# B&R Automation Studio project IecStringPrj
Automation Studio 4.11.5.46 SP; Sample project and development for IecString library

## Configuration ARM

CPU X20CP0484, AutomationRuntime 6.3.4, Build 11.3.0

### Task classes (Cpu.sw)
```
Libraries: IecString, AsBrStr, astime, runtime
```

### Hardware
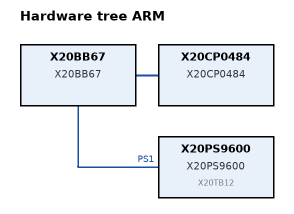
```
X20BB67 : X20BB67 v1.3.1.0
X20CP0484 : X20CP0484 v1.8.1.0  [SL -> X20BB67.SL1]
  Connector IF2:
    ActivateDevice = 1
    InaPort = 11160
  ConfigurationID = IecStringProject_ARM
  UserPartitionSize = 0
  TimerDeviceType = SWIOTIMER
  Cyclic1Duration = 10000
  Cyclic1Tolerance = 10000
  Cyclic2Duration = 20000
  Cyclic2Tolerance = 20000
  Cyclic3Duration = 50000
  Cyclic3Tolerance = 50000
  Cyclic4Duration = 100000
  Cyclic4Tolerance = 100000
  Cyclic5Duration = 200000
  Cyclic5Tolerance = 200000
  Cyclic6Duration = 500000
  Cyclic6Tolerance = 500000
  Cyclic7Duration = 1000000
  Cyclic7Tolerance = 1000000
  Cyclic8Duration = 10000
  Cyclic8Tolerance = 30000000
  FileDevice1
  FileDeviceName1 = USER
  FileDevicePath1 = USER_PATH
  ActivateFtpServer = 1
  ActivateWebServer = 1
  ActivateSdm = 1
X20PS9600 : X20PS9600 v1.6.2.0  [PS -> X20BB67.PS1; SS1 -> X20TB12.SS]
X20TB12 : X20TB12 v1.0.0.0
```

## Configuration ARsim

CPU PC_any, AutomationRuntime B4.73, Build 4.1.2, Vc V4.72.2

### Task classes (Cpu.sw)
```
Cyclic#1:
  Sample <- Sample.prg
Binaries: FWRules, TCData, udbdef, asfw, User, iomap, sysconf, arconfig, ashwd, Role, ashwac
Libraries: BRSE_ARL, AsBrStr, ArEventLog, sys_lib, runtime, asieccon, astime, IecFrmtStr
```

## Configuration Hardware

CPU X20CP1585, AutomationRuntime E4.92, Build 6.3.0

### Task classes (Cpu.sw)
```
Cyclic#1:
  ACopy1C <- Source.Performance.ACopy1C.prg
  ACopy2Iec <- Source.Performance.ACopy2Iec.prg
  ACopy3Brs <- Source.Performance.ACopy3Brs.prg
  ACopy4Lib <- Source.Performance.ACopy4Lib.prg
  PerfCCopy <- (binary)
  PerfBrCopy <- (binary)
  PerfISDec <- (binary)
  PerfBrDec <- (binary)
  PerfISCopy <- (binary)
Libraries: IecString, AsBrStr, astime, runtime
```

### Hardware
```
X20CP1585 : X20CP1585 v1.10.0.0
  Connector IF1:
    ActivateIna = 0
  Connector IF2:
    ActivateDevice = 1
    HostName = chicago-x20cp1585
  Connector IF3:
    EplHostName = chicago-x20cp1585
    HostName = chicago-x20cp1585
  ConfigurationID = IecStringProject_Hardware
  FileDevice1
  FileDeviceName1 = USER
  FileDevicePath1 = USER_PATH
  EthernetHostName = chicago-x20cp1585
```

## Configuration IA32

CPU X20CP1685, AutomationRuntime 6.3.4, Build 11.3.0, Vc 

### Task classes (Cpu.sw)
```
Libraries: IecString
```

### Hardware
```
X20CP1685 : X20CP1685 v1.8.1.0
  FileDevice1
  FileDeviceName1 = USER
  FileDevicePath1 = USER_PATH
```

## Configuration Intel

CPU X20CP1586, AutomationRuntime E4.92, Build 6.3.0

### Task classes (Cpu.sw)
```
Cyclic#1:
  PerfCCopy <- (binary)
  PerfBrCopy <- (binary)
  PerfISDec <- (binary)
  PerfBrDec <- (binary)
  PerfISCopy <- (binary)
Binaries: TCData, udbdef, asfw, sysconf, arconfig, ashwd, ashwac
Libraries: IecString, astime, standard, asieccon
```

### Hardware
```
X20CP1586 : X20CP1586 v1.10.0.0
  Connector IF1:
    ActivateIna = 0
  Connector IF2:
    ActivateDevice = 1
  ConfigurationID = IecStringProject_Intel
  FileDevice1
  FileDeviceName1 = USER
  FileDevicePath1 = USER_PATH
```

## Configuration Simulation

CPU PC_any, AutomationRuntime C4.90, Build 4.1.2, Vc 

### Task classes (Cpu.sw)
```
Cyclic#1:
  Sample <- Sample.prg
  CUsage <- CUsage.prg
Binaries: FWRules, TCData, udbdef, asfw, User, iomap, sysconf, arconfig, ashwd, Role, ashwac
Libraries: AsBrStr, runtime, IecString, asieccon, astime
```

### Hardware
```
X20CP1586 : X20CP1586 v1.10.0.0
  Connector IF1:
    ActivateIna = 0
  Connector IF2:
    ActivateDevice = 1
    InaPort = 11160
  ConfigurationID = IecStringPrj_Simulation
```

## Configuration UnitTest

CPU PC_any, AutomationRuntime 6.3.4, Build 11.3.0

### Task classes (Cpu.sw)
```
Cyclic#1 (cycle 1000 us):
  TestSuite <- Source.UnitTest.TestSuite.prg
  ExSplit <- Source.Example.ExSplit.prg
Binaries: udbdef, TCData, sysconf, ashwd, asfw, arconfig, ashwac
Libraries: IecString, runtime, astime, UnitTest, UtMgr, sys_lib, UtWs, AsIecCon, AsBrStr
```

### Hardware
```
PC : PC_any v1.1.2.0 (OrderNumber=PC)
  ConfigurationID = IecStringProject_UnitTest
  SystemTick = 1000
  Cyclic1Duration = 1000
  FileDevice1
  FileDeviceName1 = USER
  FileDevicePath1 = USER_PATH
  ActivateFtpServer = 1
  ActivateWebServer = 1
  WebServerProtocol = 1
  ActivateSdm = 1
```

## Configuration X20CPU

CPU X20CP1585, AutomationRuntime E4.92, Build 6.3.0

CPU X20CP1586, AutomationRuntime E4.92, Build 4.1.2, Vc 

### Task classes (Cpu.sw)
```
Cyclic#1:
  CPUCopy <- Source.Performance.CPUCopy.prg
Cyclic#4:
  TestSuite <- Source.UnitTest.TestSuite.prg
  IECST <- Source.Sample.IECST.prg
  TestCStr <- Source.Compare.TestCStr.prg
Libraries: AsBrStr, IecString, UnitTest, UtMgr, UtWs, AsARCfg, runtime, AsIecCon, astime, sys_lib
```

### Task classes (Cpu.sw)
```
Cyclic#4:
  TestSuite <- TestSuite.prg
  IECST <- IECST.prg
Libraries: AsBrStr, IecString, UnitTest, UtMgr, UtWs, AsARCfg, runtime, AsIecCon, astime, sys_lib
```

### Hardware
```
X20CP1585 : X20CP1585 v1.10.0.0
  Connector IF1:
    ActivateIna = 0
  Connector IF2:
    ActivateDevice = 1
    HostName = chicago-x20cp1585
    InaPort = 11160
  Connector IF3:
    EplHostName = chicago-x20cp1585
    HostName = chicago-x20cp1585
  ConfigurationID = IecStringProject_X20CPU
  FileDevice1
  FileDeviceName1 = USER
  FileDevicePath1 = USER_PATH
  EthernetHostName = chicago-x20cp1585
```

## Logical view

Binary libraries used (declarations not repeated): IecString, UnitTest, UtMgr, UtWs, runtime, sys_lib, astime, AsBrStr, standard, AsIecCon

### Package Logical/Libraries - Global libraries

### Library Logical/Libraries/BRSE_ARL (ANSIC, version 2.00.0)
Depends on: AsBrStr, SYS_Lib, ArEventLog

#### BRSE_ARL.fun
```iecst
FUNCTION BRSE_ARL_Alloc : UINT (*Allocates the FIFO buffer for the logger*)
	VAR_INPUT
		ID : UINT; (*Logger ID of the logbook to be written to*)
		Name : STRING[25]; (*Name of the logbook to which to write to.*)
		LogbookSize : UDINT; (*Size of the logbook in bytes (if a new one has to be created).*)
		MessageSize : UDINT; (*Maximum length of a single message string for the logbook*)
		BufferedEntries : UDINT; (*Maximum number of messages that can be stored in the FIFO buffer*)
	END_VAR
END_FUNCTION
(*	VAR_INPUT
		ID : UINT; (*Logger ID of the logbook to be written to*)
(*		ErrorNumber : UDINT; (*Error number to show up in the logbook*)
(*FUNCTION BRSE_ARL_Info : UINT (*Writes an info message to the logbook*)
(*		ErrorMessage : STRING[32767]; (*Error message in the logbook*)
(*		pMsgData : UDINT; (*Address of a BRSE_ARL_Arguments_typ structure that contains data values*)
(*	END_VAR
END_FUNCTION--*/ *)

FUNCTION BRSE_ARL_Cyclic : DINT (*Cyclic call to flush pending entries to the logbook*)
	VAR_INPUT
		ID : UINT; (*Logger ID of the logbook to be written to*)
	END_VAR
END_FUNCTION

FUNCTION_BLOCK BRSE_ARL_DebugInfo
	VAR_INPUT
		ID : UINT;
	END_VAR
	VAR_OUTPUT
		Info : BRSE_ARL_Logger_typ;
		Status : UINT;
	END_VAR
END_FUNCTION_BLOCK
(*FUNCTION BRSE_ARL_Fatal : UINT (*Writes a fatal message to the logbook*)
(*	VAR_INPUT
				ID : UINT; (*Logger ID of the logbook to be written to*)
(*		ErrorNumber : UDINT; (*Error number to show up in the logbook*)
(*		ErrorMessage : STRING[32767]; (*Error message in the logbook*)
(*		pMsgData : UDINT; (*Address of a BRSE_ARL_Arguments_typ structure that contains data values*)
(*	END_VAR
(*END_FUNCTION *)

FUNCTION BRSE_ARL_Free : UINT (*Deallocates the FIFO buffer *)
	VAR_INPUT
		ID : UINT; (*Logger ID of the logbook to be written to*)
	END_VAR
END_FUNCTION
(*FUNCTION BRSE_ARL_Warning : UINT (*Writes a warning message to the logbook*)
(*	VAR_INPUT
		ID : UINT; (*Logger ID of the logbook to be written to*)
(*		ErrorNumber : UDINT; (*Error number to show up in the logbook*)
(*		ErrorMessage : STRING[32767]; (*Error message in the logbook*)
(*		pMsgData : UDINT; (*Address of a BRSE_ARL_Arguments_typ structure that contains data values*)
(*	END_VAR
(*END_FUNCTION*)

FUNCTION BRSE_ARL_Log : UINT
	VAR_INPUT
		ID : UINT;
		ErrorNumber : UDINT;
		User : STRING[32];
		ErrorMessage : STRING[32767];
	END_VAR
END_FUNCTION
```

#### BRSE_ARL.typ
```iecst
TYPE
	BRSE_ARL_Arguments_typ : 	STRUCT
		r : ARRAY[0..4]OF REAL;
		s : ARRAY[0..4]OF UDINT;
		b : ARRAY[0..4]OF BOOL;
		i : ARRAY[0..4]OF DINT;
	END_STRUCT;
	BRSE_ARL_Logger_typ : 	STRUCT  (* ID CHECK *)
		ID : UDINT; (*unsigned long ID;*) (*Size of the structure*)
		LoggerTypSize : DINT; (*long LoggerTypSize;*) (*VARIABLES*)
		LogbookIdent : UDINT; (*UDINT LogbookIdent;*)
		LogbookSize : UDINT; (*UDINT LogbookSize;*) (*Size of the logbook*)
		LogbookName : STRING[26]; (*char LogbookName[26];*) (*Name of the logbook (max. 25 chars)*)
		MaxMessageSize : UDINT; (*unsigned int MaxMessageSize;*) (*Max. size of a text message*)
		Cyclic_Step : UDINT; (*unsigned int Cyclic_Step;*) (* FUNCTION BLOCKS *)
		FB_ArEventLogGetIdent : ArEventLogGetIdent; (*AsArLogGetInfo_typ FB_AsArLogGetInfo;*)
		FB_ArEventLogCreate : ArEventLogCreate; (*AsArLogCreate_typ  FB_AsArLogCreate;*)
		FB_ArEventLogWrite : ArEventLogWrite; (*AsArLogWrite_typ   FB_AsArLogWrite;*) (*FIFO BUFFER*)
		fifo_write_lock : BOOL; (*Locks critical sections in the FIFO write processing*)
		fifo_reset : BOOL; (*Clearing FIFO memory, used if FIFO full when trying to read.*)
		tempString : STRING[50];
		EntrySize : UDINT; (* Size of a single logbook entry *)
		MaxBufEntries : UDINT; (*Max. number of buffered entries*)
		CurBufEntries : UDINT; (*Number of entries in the buffer*)
		ReadIndex : UDINT; (*Current index from which to read*)
		WriteIndex : UDINT; (* Current index at which to write *)
		Buffer : ARRAY[0..0]OF BRSE_ARL_LogbookEntry_typ; (*Buffer start position (must be last in the struct)*)
	END_STRUCT;
	BRSE_ARL_LogbookEntry_typ : 	STRUCT
		User : STRING[36];
		ErrorNo : UDINT;
		ErrorMsg : STRING[0]; (* Only buffer start position, size depends on the requested size in Alloc *)
	END_STRUCT;
END_TYPE
```

#### brse_arl_alloc.c
```c
/*! \file brse_arl_alloc.c */

#include "brse_arl_main.h"

/* List of all available loggers */
BRSE_ARL_Logger_typ* BRSE_ARL_LoggerList[BRSE_ARL_MAX_LOGGERS];

/*! \interface BRSE_ARL_Alloc
	\brief Allocates the FIFO buffer for the logger

	This function allocates a FIFO buffer of the given size to be used for further
	buffered logbook writing functions. It also takes parameters that will be used in \ref BRSE_ARL_Cyclic().
	NOTE: Should be called in the _INIT part of a task!

	The following is done in \ref BRSE_ARL_Cyclic(): If logbook does not exist a new one will be created with the supplied name.
	If no name has been supplied, the default user logbook will be used.

	\param ID Logger ID of the logbook to be written to
    \param Name Name of the logbook to which to write to.
    \param LogbookSize Size of the logbook in bytes (if a new one has to be created). Note: at least 4096
    \param MessageSize Maximum length of a single message string for the logbook
    \param BufferedEntries Maximum number of messages that can be stored in the FIFO buffer
    \retval \c 0 Function call successful
*/
unsigned short BRSE_ARL_Alloc(unsigned short ID, plcstring* Name, unsigned long LogbookSize, unsigned long MessageSize, unsigned long BufferedEntries)
{
	BRSE_ARL_Logger_typ* pLogger;
	unsigned long EntrySize;
	unsigned long LoggerTypSize;

	/* Check if ID is in range */
	if (ID >= BRSE_ARL_MAX_LOGGERS)
	{
		return BRSE_ARL_ID_NOT_VALID;
	}

	/* Access the chosen logger */
	pLogger = BRSE_ARL_LoggerList[ID];

	/* Check, if ID is valid */
	if ((pLogger != NULL) && (pLogger->ID == (BRSE_ARL_ID_BASE | (unsigned long)ID)))
	{
		return BRSE_ARL_ID_ALREADY_INITIALIZED;
	}

	/* ID is not used yet, so allocate memory for it */

	/* Calculate the entry size and the logger size */
	EntrySize = (unsigned long)sizeof(BRSE_ARL_LogbookEntry_typ) + MessageSize + 1;
	LoggerTypSize = (unsigned long)sizeof(BRSE_ARL_Logger_typ) + BufferedEntries * EntrySize;

	/* Allocate memory for the logger */
	if (TMP_alloc(LoggerTypSize, (void**)&pLogger) != 0)
	{
		/* Memory allocation failed */
		return BRSE_ARL_OUT_OF_MEMORY;
	}
	/* Put valid information into the logger structure */
	memset((void*)pLogger, 0, LoggerTypSize);

	/* Store some information */
	pLogger->ID = BRSE_ARL_ID_BASE | (unsigned long)ID;
	pLogger->LoggerTypSize = LoggerTypSize;

	strncpy(pLogger->LogbookName, Name, sizeof(pLogger->LogbookName));
	pLogger->LogbookSize = LogbookSize;
	pLogger->MaxMessageSize = MessageSize;
	pLogger->EntrySize = EntrySize;
	pLogger->MaxBufEntries = BufferedEntries;

	/* Save the new logger */
	BRSE_ARL_LoggerList[ID] = pLogger;

	return ERR_OK;
}

/*! \interface BRSE_ARL_Free
	\brief Deallocates the FIFO buffer

	This function writes all pending entries to the logbook and closes down the buffer.
	NOTE: Not to be called in the cyclic part of a task!

	\param ID Logger ID of the logbook to be written to
    \return \c 0 Function call successful
*/
unsigned short BRSE_ARL_Free(unsigned short ID)
{
	/* Check if ID is valid */
	if ((ID >= BRSE_ARL_MAX_LOGGERS)
		|| (BRSE_ARL_LoggerList[ID] == NULL)
		|| (BRSE_ARL_LoggerList[ID]->ID != (BRSE_ARL_ID_BASE | (unsigned long)ID)))
	{
		return BRSE_ARL_ID_NOT_VALID;
	}

	/* Flush pending writes */
	while (BRSE_ARL_Cyclic(ID) == 65535);

	/* Release allocated memory */
	TMP_free(BRSE_ARL_LoggerList[ID]->LoggerTypSize, (void*)BRSE_ARL_LoggerList[ID]);
	BRSE_ARL_LoggerList[ID] = NULL;

	return ERR_OK;
}
```

#### brse_arl_cyclic.c
```c
/*! \file brse_arl_cyclic.c */

#include "brse_arl_main.h"

/*! \interface BRSE_ARL_Cyclic
	\brief Cyclic call to flush pending entries to the logbook

	This function writes pending entries to the logbook and has to be called cyclically.

	\param ID Logger ID of the logbook to be written to
    \retval 0 all messages written to logger
	\retval 65535 pending entries to be written
	\retval Error Error code from the ArEventLog library
*/

long BRSE_ARL_Cyclic(unsigned short ID)
{
	BRSE_ARL_Logger_typ* pLogger = NULL;
	BRSE_ARL_LogbookEntry_typ* pCurEntry = NULL;
	DINT status = ERR_FUB_BUSY;

	/* Check if ID is valid */
	if ((ID >= BRSE_ARL_MAX_LOGGERS)
		|| (BRSE_ARL_LoggerList[ID] == NULL)
		|| (BRSE_ARL_LoggerList[ID]->ID != (BRSE_ARL_ID_BASE | (unsigned long)ID)))
	{
		return BRSE_ARL_ID_NOT_VALID;
	}

	/* Access the chosen logger */
	pLogger = BRSE_ARL_LoggerList[ID];

	switch (pLogger->Cyclic_Step)
	{
		/* Initialize */
		case 0:

			pLogger->Cyclic_Step = 1;

		/* GET LOGBOOK */
		case 1:
			/* Check if a logbook with the given name is existing */
			pLogger->FB_ArEventLogGetIdent.Execute = TRUE;
			strcpy(pLogger->FB_ArEventLogGetIdent.Name, pLogger->LogbookName);

			ArEventLogGetIdent(&pLogger->FB_ArEventLogGetIdent);

			if(pLogger->FB_ArEventLogGetIdent.Done)
			{
				/* Save the ident of the exisiting logbook */
				pLogger->LogbookIdent = pLogger->FB_ArEventLogGetIdent.Ident;

				/* Go to operating state */
				pLogger->Cyclic_Step = 10;
				status = ERR_FUB_BUSY;
			}
			else if(pLogger->FB_ArEventLogGetIdent.Error)
			{
				if(pLogger->FB_ArEventLogGetIdent.StatusID == arEVENTLOG_ERR_LOGBOOK_NOT_FOUND)
				{
					pLogger->Cyclic_Step = 2;
					status = ERR_FUB_BUSY;
				}
				else
				{
					status = pLogger->FB_ArEventLogGetIdent.StatusID;
				}
			}
			else
			{
				status = ERR_FUB_BUSY;
			}

			break;

		/* CREATE LOGBOOK */
		case 2:
			/* Create a new logbook in USRROM */
			pLogger->FB_ArEventLogCreate.Execute = TRUE;
			strcpy(pLogger->FB_ArEventLogCreate.Name, pLogger->LogbookName);
			pLogger->FB_ArEventLogCreate.Size = pLogger->LogbookSize;
			pLogger->FB_ArEventLogCreate.Persistence = arEVENTLOG_PERSISTENCE_PERSIST;

			ArEventLogCreate(&pLogger->FB_ArEventLogCreate);

			if(pLogger->FB_ArEventLogCreate.Done)
			{
				pLogger->LogbookIdent = pLogger->FB_ArEventLogCreate.Ident;

				/* Go to operating state */
				pLogger->Cyclic_Step = 10;
				status = ERR_FUB_BUSY;
			}
			else if(pLogger->FB_ArEventLogCreate.Busy)
			{
				status = ERR_FUB_BUSY;
			}
			else if(pLogger->FB_ArEventLogCreate.Error)
			{
				status = pLogger->FB_ArEventLogCreate.StatusID;
			}

			break;

		/* POP ENTRY FROM THE FIFO AND WRITE IT TO THE LOGBOOK */
		case 10:
			status = ERR_FUB_BUSY;
			if ( (pLogger->CurBufEntries == 0) )
			{
				/* No entry in the fifo */
				/* Answer with OK then... */
				status = ERR_OK;
			}
			else if (!pLogger->fifo_write_lock)
			{
				if ( (pLogger->CurBufEntries >= pLogger->MaxBufEntries) )
				{
					/*Lock the buffer directly to avoid loosing data*/
					pLogger->fifo_reset = 1;

					/*State change, prepare to reset buffer*/
					pLogger->Cyclic_Step = 14;

					status = ERR_FUB_BUSY;

				}
				else
				{
					/* Got an entry in the fifo */
					pCurEntry = (BRSE_ARL_LogbookEntry_typ*)((void*)pLogger->Buffer + pLogger->EntrySize * pLogger->ReadIndex);

					pLogger->FB_ArEventLogWrite.Execute = TRUE;
					pLogger->FB_ArEventLogWrite.Ident = pLogger->LogbookIdent;
					pLogger->FB_ArEventLogWrite.EventID = pCurEntry->ErrorNo;
					pLogger->FB_ArEventLogWrite.AddDataSize = strlen(pCurEntry->ErrorMsg) + 1;
					pLogger->FB_ArEventLogWrite.AddDataFormat = arEVENTLOG_ADDFORMAT_TEXT;
					pLogger->FB_ArEventLogWrite.AddData = (UDINT)pCurEntry->ErrorMsg;
					strcpy(pLogger->FB_ArEventLogWrite.ObjectID, pCurEntry->User);

					if(pLogger->FB_ArEventLogWrite.Done)
					{
						pLogger->FB_ArEventLogWrite.Execute = FALSE;
					}

					ArEventLogWrite(&pLogger->FB_ArEventLogWrite);

					if(pLogger->FB_ArEventLogWrite.Done)
					{
						pLogger->ReadIndex++;
						if (pLogger->ReadIndex >= pLogger->MaxBufEntries)
						{
							pLogger->ReadIndex = 0;
						}

						pLogger->CurBufEntries--;

						/* Return OK if no more entries shall be written */
						status = (pLogger->CurBufEntries == 0) ? ERR_OK : ERR_FUB_BUSY;
					}
					else if(pLogger->FB_ArEventLogWrite.Error)
					{
						status = pLogger->FB_ArEventLogWrite.StatusID;
					}
					else
					{
						status = ERR_FUB_BUSY;
					}
				}
			}
			else
			{
				/* Write is active */
				status = ERR_FUB_BUSY;
			}
			break;
		case 14:
			status = ERR_FUB_BUSY;

			if (pLogger->FB_ArEventLogWrite.StatusID == ERR_FUB_BUSY )
			{
				/*Wait if a line is being written to the logg book.*/
				ArEventLogWrite(&pLogger->FB_ArEventLogWrite);

			}
			else
			{

				/*Switch state, empty buffer.*/
				pLogger->Cyclic_Step = 15;
			}

			break;

		case 15: /*Output reset start message*/
				status = ERR_FUB_BUSY;

				pLogger->FB_ArEventLogWrite.Execute 		= TRUE;
				pLogger->FB_ArEventLogWrite.Ident 			= pLogger->LogbookIdent;
				pLogger->FB_ArEventLogWrite.EventID 		= -536820909; /* Severity = Error, Code = 50003 */
				strcpy(pLogger->tempString, "BUFFER RESET STARTED");
				pLogger->FB_ArEventLogWrite.AddData			= (UDINT)(pLogger->tempString);
				pLogger->FB_ArEventLogWrite.AddDataSize 	= strlen(pLogger->tempString) + 1;
				pLogger->FB_ArEventLogWrite.AddDataFormat 	= arEVENTLOG_ADDFORMAT_TEXT;

				ArEventLogWrite(&pLogger->FB_ArEventLogWrite);

				if (pLogger->FB_ArEventLogWrite.StatusID == ERR_OK )
				{
					/*Switch state, empty buffer.*/
					pLogger->Cyclic_Step = 20;

				}
			break;

		case 20: /*Empty the buffer, reset.*/
			status = ERR_FUB_BUSY;
			if ( (pLogger->CurBufEntries == 0) )
			{
				/*Buffer reset completed, switcht to state where message is output.*/
				pLogger->Cyclic_Step = 21;

			}
			else
			{
				/*Empty buffer*/
				/* Got an entry in the fifo */
				pCurEntry = (BRSE_ARL_LogbookEntry_typ*)((UDINT)pLogger->Buffer + pLogger->EntrySize * pLogger->ReadIndex);

				pLogger->FB_ArEventLogWrite.Execute 		= TRUE;
				pLogger->FB_ArEventLogWrite.Ident 			= pLogger->LogbookIdent;
				pLogger->FB_ArEventLogWrite.EventID 		= pCurEntry->ErrorNo;
				//TODO: Event ID log level
				pLogger->FB_ArEventLogWrite.AddDataFormat 	= arEVENTLOG_ADDFORMAT_TEXT;
				pLogger->FB_ArEventLogWrite.AddData 		= (UDINT)pCurEntry->ErrorMsg;
				strcpy(pLogger->FB_ArEventLogWrite.ObjectID, pCurEntry->User);
				//					pLogger->FB_AsArLogWrite.mem = (UDINT)NULL;
				//					pLogger->FB_AsArLogWrite.len = 0;

				ArEventLogWrite(&pLogger->FB_ArEventLogWrite);

				if(pLogger->FB_ArEventLogWrite.Done)
				{
					pLogger->ReadIndex++;
					if (pLogger->ReadIndex >= pLogger->MaxBufEntries)
					{
						pLogger->ReadIndex = 0;
					}

					pLogger->CurBufEntries--;

					/* Return OK if no more entries shall be written */
					status = (pLogger->CurBufEntries == 0) ? ERR_OK : ERR_FUB_BUSY;
				}
				else if(pLogger->FB_ArEventLogWrite.Error)
				{
					status = pLogger->FB_ArEventLogWrite.StatusID;
				}
				else
				{
					status = ERR_FUB_BUSY;
				}
			}
			break;

		case 21: /*Output message the reset is completed*/
				status = ERR_FUB_BUSY;

				pLogger->FB_ArEventLogWrite.Execute 		= TRUE;
				pLogger->FB_ArEventLogWrite.Ident 			= pLogger->LogbookIdent;
				pLogger->FB_ArEventLogWrite.EventID			= -536820908;
				pLogger->FB_ArEventLogWrite.AddDataFormat 	= arEVENTLOG_ADDFORMAT_TEXT;
				strcpy(pLogger->tempString, "BUFER RESET COMPLETED");
				pLogger->FB_ArEventLogWrite.AddData 		= (UDINT)pLogger->tempString;
				pLogger->FB_ArEventLogWrite.AddDataSize 	= strlen(pLogger->tempString) + 1;

				ArEventLogWrite(&pLogger->FB_ArEventLogWrite);

				status = ERR_FUB_BUSY;
				if (pLogger->FB_ArEventLogWrite.StatusID == ERR_OK )
				{
					status = ERR_OK;
					pLogger->fifo_reset = 0;
					pLogger->Cyclic_Step = 10;

				}

			break;

	}

	return status;
}
```

#### brse_arl_log.c
```c
/*! \file brse_arl_log.c */

#include "brse_arl_main.h"

/* Internal function to concat the string */
//static void CreateErrorMessage(char* dst, long dst_size, char* src, BRSE_ARL_Arguments_typ* pArguments)
//{
//	/* Temporary array for string concatenations */
//	char temp_string[16];
//
//	/* Size of a string that is concatenated to the destination */
//	int concat_string_size;
//
//	/* Array index counters */
//	int bool_counter   = 0;
//	int int_counter    = 0;
//	int real_counter   = 0;
//	int string_counter = 0;
//
//	/* Run through the source message and copy it to the destination until src is empty or destination is full */
//	while ((*src != '\0') && (dst_size > 0))
//	{
//		/* Special character found and MessageData given */
//		if ((pArguments != NULL) && (*src == '%'))
//		{
//			/* Temporary 'close' the destination string (to allow strcat...) */
//			*dst = '\0';
//
//			/* Consume the char and investigate the command */
//			switch (*(++src))
//			{
//				/* Insert bool */
//				case 'b':
//					/* Only take a value if an array entry exists */
//					if (bool_counter < ARRAY_ENTRIES(pArguments->b))
//					{
//						if (pArguments->b[bool_counter])
//						{
//							strncat(dst, "TRUE", dst_size);
//							concat_string_size = MIN(dst_size, 4);
//						}
//						else
//						{
//							strncat(dst, "FALSE", dst_size);
//							concat_string_size = MIN(dst_size, 5);
//						}
//						bool_counter++;
//						dst += concat_string_size;
//						dst_size -= concat_string_size;
//					}
//					src++;
//					break;
//
//				/* Insert integer */
//				case 'i':
//					/* Only take a value if an array entry exists */
//					if (int_counter < ARRAY_ENTRIES(pArguments->i))
//					{
//						concat_string_size = brsitoa(pArguments->i[int_counter], (UDINT)temp_string);
//						concat_string_size = MIN(dst_size, concat_string_size);
//						strncat(dst, temp_string, dst_size);
//						int_counter++;
//						dst += concat_string_size;
//						dst_size -= concat_string_size;
//					}
//					src++;
//					break;
//
//				/* Insert real */
//				case 'r':
//					/* Only take a value if an array entry exists */
//					if (real_counter < ARRAY_ENTRIES(pArguments->r))
//					{
//						concat_string_size = brsftoa(pArguments->r[real_counter], (UDINT)temp_string);
//						concat_string_size = MIN(dst_size, concat_string_size);
//						strncat(dst, temp_string, dst_size);
//						real_counter++;
//						dst += concat_string_size;
//						dst_size -= concat_string_size;
//					}
//					src++;
//					break;
//
//				/* Insert string */
//				case 's':
//					/* Only take a value if an array entry exists */
//					if (string_counter < ARRAY_ENTRIES(pArguments->s))
//					{
//						if (pArguments->s[string_counter])
//						{
//							strncat(dst, (char*)pArguments->s[string_counter], dst_size);
//							concat_string_size = MIN(dst_size, strlen((char*)pArguments->s[string_counter]));
//							dst += concat_string_size;
//							dst_size -= concat_string_size;
//						}
//						string_counter++;
//					}
//					src++;
//					break;
//
//				/* Insert percent */
//				case '%':
//					*dst++ = '%';
//					src++;
//					dst_size--;
//					break;
//
//				/* ELSE */
//				default:
//					/* Ignore the character */
//					src++;
//					break;
//			}
//		}
//		else
//		{
//			*dst++ = *src++;
//			dst_size--;
//		}
//	}
//
//	/* Add the end of string */
//	*dst = '\0';
//}
/*! \interface BRSE_ARL_Log
	\brief Writes a message to the logbook

	This function writes a message to the buffered logbook using the given
	ErrorNumber and ErrorMessage. If you add your own error number be sure that the customer bit is set.
	USE 32-bit event ID to make error numbers - ArEventLogMakeEventID()

	If the address of a BRSE_ARL_Arguments_typ structure is passed,
	its variables can be referenced in the ErrorMessage string by %[b|i|r|s]. Each usage
	of a wildcard consumes the according variable and moves on the next one within the array.

	E.g:
	MessageString = "Digital input %s: %b, analogue input %s: %i"
	BRSE_ARL_Arguments_typ = { s[0] = "Valve 1"; s[1] = "Encoder 2"; b[0] = 'TRUE'; i[0] = 4388 }

	Will create a logbook entry:
	"Digital input Valve 1: TRUE, analogue input Encoder 2: 4388"

	@ref Examples

	\param ID Logger ID of the logbook to be written to
    \param ErrorNumber Error number to show up in the logbook
    \param User Created by to show up in the logbook
    \param ErrorMessage Error message in the logbook
    \param pArguments Address of a BRSE_ARL_Arguments_typ structure that contains data values
    \retval 0 Function call successful
*/
unsigned short BRSE_ARL_Log(unsigned short ID,unsigned long ErrorNumber,plcstring* User, plcstring* ErrorMessage)
{
	BRSE_ARL_Logger_typ* pLogger;
	BRSE_ARL_LogbookEntry_typ* pCurEntry;
	UINT status;

	/* Check the ID */
	if ((ID >= BRSE_ARL_MAX_LOGGERS)
		|| (BRSE_ARL_LoggerList[ID] == NULL)
		|| (BRSE_ARL_LoggerList[ID]->ID != (BRSE_ARL_ID_BASE | (unsigned long)ID)))
	{
		return BRSE_ARL_ID_NOT_VALID;
	}

	/* Access the chosen logger */
	pLogger = BRSE_ARL_LoggerList[ID];

	/* Check and set the semaphore */
	if (!pLogger->fifo_write_lock && !pLogger->fifo_reset)
	{
		pLogger->fifo_write_lock = TRUE;

		/* Create the logbook message and put it into the buffer */
		pCurEntry = (BRSE_ARL_LogbookEntry_typ*)((UDINT)pLogger->Buffer + pLogger->EntrySize * pLogger->WriteIndex);

		strcpy(pCurEntry->User, User);
		pCurEntry->ErrorNo = ErrorNumber;
		strcpy(pCurEntry->ErrorMsg, ErrorMessage); /* Copy the error message string as is */

		/* Do not format the error message here any more */
		//CreateErrorMessage(pCurEntry->ErrorMsg, (long)pLogger->MaxMessageSize, ErrorMessage,(BRSE_ARL_Arguments_typ*)pArguments);

		/* Adjust the FIFO:
	     * Increase the WriteIndex, but reset it to 0 if MaxBufEntries have been exceeded
		 */
		pLogger->WriteIndex++;
		if (pLogger->WriteIndex >= pLogger->MaxBufEntries)
		{
			pLogger->WriteIndex = 0;
		}

		/* Check if space is available in the buffer */
		if (pLogger->CurBufEntries >= pLogger->MaxBufEntries)
		{
			/*buffer is full, shift the read position (delete the oldest entry)*/
			pLogger->ReadIndex++;
			if (pLogger->ReadIndex >= pLogger->MaxBufEntries)
			{
				pLogger->ReadIndex = 0;
			}
		}
		else
		{
			/*buffer is not yet full, increase the buffer size*/
			pLogger->CurBufEntries++;
		}

		pLogger->fifo_write_lock = FALSE;
		status = ERR_OK;
	}
	else
	{
		status = ERR_FUB_BUSY;
	}

	return status;
}

/*! \interface BRSE_ARL_Info
	\brief Writes an info message to the logbook

	This function writes an info message to the buffered logbook using the given
	ErrorNumber and ErrorMessage. If you add your own error number be sure to only
	use values > 50000, lower values are reserved for AS.

	If the address of a BRSE_ARL_Arguments_typ structure is passed,
	its variables can be referenced in the ErrorMessage string by %[b|i|r|s]. Each usage
	of a wildcard consumes the according variable and moves on to the next one within the array.

	E.g:
	MessageString = "Digital input %s: %b, analogue input %s: %i"
	BRSE_ARL_Arguments_typ = { s[0] = "Valve 1"; s[1] = "Encoder 2"; b[0] = 'TRUE'; i[0] = 4388 }

	Will create a logbook entry:
	"Digital input Valve 1: TRUE, analogue input Encoder 2: 4388"

	@ref Examples

	\param ID Logger ID of the logbook to be written to
    \param ErrorNumber Error number to show up in the logbook
    \param ErrorMessage Error message in the logbook
    \param pArguments Address of a BRSE_ARL_Arguments_typ structure that contains data values
    \retval 0 Function call successful
*/
//unsigned short BRSE_ARL_Info(unsigned short ID, unsigned long ErrorNumber, plcstring* ErrorMessage, unsigned long pArguments)
//{
//	return BRSE_ARL_Log(ID, 1, ErrorNumber, ErrorMessage, (BRSE_ARL_Arguments_typ*)pArguments);
//}

/*! \interface BRSE_ARL_Warning
	\brief Writes a warning message to the logbook

	This function writes a warning message to the buffered logbook using the given
	ErrorNumber and ErrorMessage. If you add your own error number be sure to only
	use values > 50000, lower values are reserved for AS.

	If the address of a BRSE_ARL_Arguments_typ structure is passed,
	its variables can be referenced in the ErrorMessage string by %[b|i|r|s]. Each usage
	of a wildcard consumes the according variable and moves on the next one within the array.

	E.g:
	MessageString = "Digital input %s: %b, analogue input %s: %i"
	BRSE_ARL_Arguments_typ = { s[0] = "Valve 1"; s[1] = "Encoder 2"; b[0] = 'TRUE'; i[0] = 4388 }

	Will create a logbook entry:
	"Digital input Valve 1: TRUE, analogue input Encoder 2: 4388"

	@ref Examples

	\param ID Logger ID of the logbook to be written to
    \param ErrorNumber Error number to show up in the logbook
    \param ErrorMessage Error message in the logbook
    \param pArguments Address of a BRSE_ARL_Arguments_typ structure that contains data values
    \retval 0 Function call successful
*/
//unsigned short BRSE_ARL_Warning(unsigned short ID, unsigned long ErrorNumber, plcstring* ErrorMessage, unsigned long pArguments)
//{
//	return BRSE_ARL_Log(ID, 2, ErrorNumber, ErrorMessage, (BRSE_ARL_Arguments_typ*)pArguments);
//}

/*! \interface BRSE_ARL_Fatal
	\brief Writes a fatal message to the logbook

	This function writes a fatal message to the buffered logbook using the given
	ErrorNumber and ErrorMessage. If you add your own error number be sure to only
	use values > 50000, lower values are reserved for AS.

	If the address of a BRSE_ARL_Arguments_typ structure is passed,
	its variables can be referenced in the ErrorMessage string by %[b|i|r|s], see examples.c

	E.g:
	MessageString = "Digital input %s: %b, analogue input %s: %i"
	BRSE_ARL_Arguments_typ = { s[0] = "Valve 1"; s[1] = "Encoder 2"; b[0] = 'TRUE'; i[0] = 4388 }

	Will create a logbook entry:
	"Digital input Valve 1: TRUE, analogue input Encoder 2: 4388"

	@ref Examples

	\param ID Logger ID of the logbook to be written to
    \param ErrorNumber Error number to show up in the logbook
    \param ErrorMessage Error message in the logbook
    \param pArguments Address of a BRSE_ARL_Arguments_typ structure that contains data values
    \retval 0 Function call successful
*/
//unsigned short BRSE_ARL_Fatal(unsigned short ID, unsigned long ErrorNumber, plcstring* ErrorMessage, unsigned long pArguments)
//{
//	return BRSE_ARL_Log(ID, 3, ErrorNumber, ErrorMessage, (BRSE_ARL_Arguments_typ*)pArguments);
//}
```

#### brse_arl_main.h
```c
/*! \file brse_arl_main.h */

/*! \mainpage BRSE_ARL
	\section Introduction
	\brief This library allows you to write to the built-in AS logbook using a set of function calls in an asynchronous way.

	The syntax of these functions is as similar as possible to the ANSI-C function "printf", as can be seen in the @ref examples.

	The asynchronous behavior is achieved by putting all incoming messages into a local circular buffer.
	This buffer stores the log messages until they are fetched by calling \ref BRSE_ARL_Cyclic() and written to the
	actual AS logbook using the built-in AS function "AsArLogWrite".

	Therefore, the synchronous nature of the "AsArLog" library is completely hidden to the user.

	\anchor buffer

	If the buffer is full when the \ref BRSE_ARL_Cyclic() function is called the buffer is automatically locked to avoid data being overwritten.
	Additionally a message is output in the logger stating "BUFFER RESET STARTED". Thereafter the buffer is emptied to the logger. When
	the buffer is empty a message stating "BUFFER RESET COMPLETED" is output into the logger and the lock of the buffer is released. The function
	\ref BRSE_ARL_Cyclic() only returns zero if the buffer is empty.

	The user must be aware that during a buffer reset new entries to the buffer can not be added which results in the possibility of having some data
	inconsistency directly after and before the buffer reset. Typically one buffer entry is lost before the reset start message. Several entries may be
	lost during the buffer reset, depending on how long time it takes to empty the buffer. Data consistency can be trusted between the reset start and
	completed messages.

	Since the library is using an circular buffer it is possible to continuously logg to the buffer in the DRAM and only dump the buffered
	data to the logger when an error occurs. This saves CPU time since the PLC does not have to transfer that data between the volatile
	and the non-volatile memory during normal operation.

	By choosing a unique ID, a specific logbook can be addressed.

	\section Overview

	\image html BRSEARLOV.jpg

	\section Description

	Start by setting up and create your logger.
	This is accomplished by the \ref BRSE_ARL_Alloc() function.
	Here you can set the name of your logger or, if a name is not given, the default user logbook will be used.
	Place \ref BRSE_ARL_Alloc() in the init part of your code.

	Next, you have to call the function \ref BRSE_ARL_Cyclic() in a cyclic way in your code to be able to "empty" the FIFO buffer
	of all its write-commands to the logbook.

	Now you can send any of the available messages to the logbook by using \ref BRSE_ARL_Fatal(), \ref BRSE_ARL_Warning(),
	or \ref BRSE_ARL_Info().

	When finished with your logbook you can use the \ref BRSE_ARL_Free() function to empty and close the FIFO buffer.
	Place \ref BRSE_ARL_Free() in the exit part of your code.

	This is an example of logbook output taken from AS.
	If you add your own error numbers, be sure to only use values > 50000, lower values are	reserved for AS.\n

	\image html LOGGBOOK.jpg
*/

#ifndef _BRSE_ARL_MAIN_H
#define _BRSE_ARL_MAIN_H

#ifndef NULL
#define NULL ((void *)0)
#endif

/* Include libraries */
#include <bur/plctypes.h>
#include <sys_lib.h>
#include <ArEventLog.h>
#include <AsBrStr.h>
#include <string.h>

/* Include internal library components */
#include "BRSE_ARL.h"

/* Logger list */
#define BRSE_ARL_MAX_LOGGERS	256
extern BRSE_ARL_Logger_typ* BRSE_ARL_LoggerList[BRSE_ARL_MAX_LOGGERS];

/* Define some basic macros */
#ifndef MIN
#define MIN(a, b) ((a) < (b) ? (a) : (b))
#endif
#ifndef MAX
#define MAX(a, b) ((a) > (b) ? (a) : (b))
#endif
#ifndef ARRAY_ENTRIES
#define ARRAY_ENTRIES(array) (sizeof(array)/sizeof(array[0]))
#endif

/* Define boolean states */
#ifndef TRUE
#define TRUE  1
#endif
#ifndef FALSE
#define FALSE 0
#endif

/* Define default error constants (if not defined before) */
#ifndef ERR_OK
#define ERR_OK                0
#endif
#ifndef ERR_FUB_ENABLE_FALSE
#define ERR_FUB_ENABLE_FALSE  65534
#endif
#ifndef ERR_FUB_BUSY
#define ERR_FUB_BUSY          65535
#endif

/* ID base value */
#define BRSE_ARL_ID_BASE 0x53450000

/* Define error constants */
#define BRSE_ARL_ID_ALREADY_INITIALIZED	58200
#define BRSE_ARL_ID_NOT_VALID 			58201
#define BRSE_ARL_BUFFER_FULL  			58202
#define BRSE_ARL_OUT_OF_MEMORY          58203

#endif
```

#### example.c
```c
/*! \page Example

	\section Example

	This example logs events in the default user logger file.

	\par LoggerExample.var:

\code

VAR
	cmdState : UINT;
	Args : BRSE_ARL_Arguments_typ;
	name : STRING[32];
	value : DINT;
	valueExceed : DINT;
	tempSet : REAL;
	tempMax : REAL;
	cooling : BOOL;
	age : INT;
END_VAR

\endcode

	\par LoggerExample.st:

\code

PROGRAM _INIT

	(*fetch the user logger module and interally address it as log 1*)
	BRSE_ARL_Alloc(1, '', 0, MessageSize:=100, BufferedEntries:=10);

	strcpy(ADR(name),ADR('Tom'));
	age := 30;

	value := 100;
	valueExceed := 12;

	tempSet := 77.3;
	tempMax := 55;
	cooling := TRUE;

END_PROGRAM

PROGRAM _CYCLIC

	CASE cmdState OF

		1: (* add an information message *)
			Args.i[0] := age;
			Args.s[0] := ADR(name);
			BRSE_ARL_Info(1, 50001, 'Your name is: %s and you are %i years old',ADR(Args));
			(*will result in:
			Your name is: Tom and you are 30 years old
			*)

		2: (*add a warning message*)
			Args.i[0] := value;
			Args.i[1] := valueExceed;
			BRSE_ARL_Warning(1, 50002, 'You have exceeded value %i by %i units',ADR(Args));
			(*will result in:
			You have exceeded value 100 by 12 units
			*)

		3: (*add a fatal message*)
			Args.r[0] := tempSet;
			Args.r[1] := tempMax;
			Args.b[0] := cooling;
			BRSE_ARL_Fatal(1, 50003, 'PLC fatal error. temperature is: %r, and cooling is %b, max temp is %r',ADR(Args));
			(*will result in:
			PLC fatal error. temperature is: 77.3, and cooling is TRUE, max temp is 55
			*)

	END_CASE

	cmdState := 0;

	(*put out the messages into the logbook*)
	BRSE_ARL_Cyclic(1);

END_PROGRAM

\endcode

The result will be the following:

\image html LoggerScreenUser.jpg

*/
```

#### version_history.c
```c
/*! \file version_history.c */

/*! \page History
\section History
\par V1.00
\arg Implemented a buffered logbook writer
\par V1.01
\arg Splitted the source file into several files
\arg renamed MsgData to Arguments, changed the String datatype to UDINT (string pointer)
\par V1.02
\arg added documentation in source files.
\arg Changed Arguments to Arguments_typ
\par V1.03
\arg Removed dependency on RtkLib
\arg Several buffered logbooks can be used (identified by a unique ID)
\par V1.04
\arg Version created for AS3.0
\par V1.05
\arg Using mystring.h instead of string.h to avoid -lc build options in the phtysical view.
\par V1.06
\arg The problem with string.h has been solved in runtime versions >= 2.95, so string.h is used instead of mystring.
\par V1.07
\arg Changed layout of the library files (in Explorer) to support AS3 library setup.
\par V1.08
\arg Changed from FIFO to circular buffer. It overwrites the oldest entry when buffer gets full, this gives the possibility
to continuously logg to the buffer and only transfer the data to the user logg when an error occurs. This uses less
CPU time then constantly writing to the user logg. Please see \ref buffer information.
\par V1.09
\arg Added new function block BRSE_ARL_DebugInfo which displays the internal stucture including the AsArLog FBs for internal usage.
\par V1.10
\arg Library dependency has been changed from AsString to AsBrStr, so that the conflictions can be avoided with ANSI-C standard functions(atof, atoi etc.)
\par V1.11
\arg Replaced (void *) with (UDINT) to avoid error in Lint
\par V1.12
\arg in function unsigned short BRSE_ARL_Cyclic(unsigned short ID) local variables are initialized
\par V1.13
\arg Much less space will be used when allocating the logger entries
\arg Logger_typ: the buffer is changed to 1 element.
\arg LoggerbookEntry_typ: the ErrorMsg is changed to 1 element.
*/
```

#### brse_arl_debuginfo.c
```c
#include "brse_arl_main.h"

void BRSE_ARL_DebugInfo(struct BRSE_ARL_DebugInfo* inst)
{
	/* Check if ID is valid */
	if ((inst->ID >= BRSE_ARL_MAX_LOGGERS)
		|| (BRSE_ARL_LoggerList[inst->ID] == NULL)
		|| (BRSE_ARL_LoggerList[inst->ID]->ID != (BRSE_ARL_ID_BASE | (unsigned long)inst->ID)))
	{
		inst->Status = BRSE_ARL_ID_NOT_VALID;
		return;
	}

	/* Copy the debug information */
 	memcpy(&inst->Info, &BRSE_ARL_LoggerList[inst->ID], sizeof(inst->Info));
	inst->Status = 0;
}
```

### Program Logical/Source/UnitTest/TestSuite (ANSIC)

#### load.c - Set loader and handler
```c
#include <UnitTest.h>

UNITTEST_TESTSET_DECLARATION copy_set;
UNITTEST_TESTSET_DECLARATION concat_set;
UNITTEST_TESTSET_DECLARATION compare_set;
UNITTEST_TESTSET_DECLARATION length_set;
UNITTEST_TESTSET_DECLARATION first_set;
UNITTEST_TESTSET_DECLARATION last_set;
UNITTEST_TESTSET_DECLARATION find_set;
UNITTEST_TESTSET_DECLARATION first_in_set;
UNITTEST_TESTSET_DECLARATION length_in_set;
UNITTEST_TESTSET_DECLARATION start_set;
UNITTEST_TESTSET_DECLARATION end_set;
UNITTEST_TESTSET_DECLARATION replace_set;
UNITTEST_TESTSET_DECLARATION split_set;
UNITTEST_TESTSET_DECLARATION format_set;
UNITTEST_TESTSET_DECLARATION decimal_set;
UNITTEST_TESTSET_DECLARATION float_set;
UNITTEST_TESTSET_DECLARATION date_time_set;

UNITTEST_TESTSET_FIXTURES (utTestSets)
{
    new_TestSet(copy_set),
    new_TestSet(concat_set),
    new_TestSet(compare_set),
    new_TestSet(length_set),
    new_TestSet(first_set),
    new_TestSet(last_set),
    new_TestSet(find_set),
    new_TestSet(first_in_set),
    new_TestSet(length_in_set),
    new_TestSet(start_set),
    new_TestSet(end_set),
    new_TestSet(replace_set),
    new_TestSet(split_set),
    new_TestSet(format_set),
    new_TestSet(decimal_set),
    new_TestSet(float_set),
    new_TestSet(date_time_set)
};

UNTITTEST_TESTSET_HANDLER();
```

#### test_copy.c - Test IecStringCopy
```c
#include <UnitTest.h>
#include <IecString.h>
#include <stdint.h>
#include <string.h>

#define SAMPLE_SIZE 81
#define SAMPLE_STRING "Hello World!"
#define LIBRARY_ERROR_NONE 0
#define LARGE_SIZE 1001

_TEST test_copy_variable(void) {
    char a[SAMPLE_SIZE], b[SAMPLE_SIZE];
    int32_t status;

    strcpy(b, SAMPLE_STRING);

    status = IecStringCopy(a, sizeof(a), b);

    TEST_ASSERT_EQUAL_STRING(SAMPLE_STRING, a);
    TEST_ASSERT_EQUAL_INT(LIBRARY_ERROR_NONE, status);

    TEST_DONE;
}

_TEST test_copy_literal(void) {
    char a[SAMPLE_SIZE];
    int32_t status;

    status = IecStringCopy(a, sizeof(a), SAMPLE_STRING);

    TEST_ASSERT_EQUAL_STRING(SAMPLE_STRING, a);
    TEST_ASSERT_EQUAL_INT(LIBRARY_ERROR_NONE, status);

    TEST_DONE;
}

_TEST test_copy_empty_source(void) {
    char a[SAMPLE_SIZE], b[SAMPLE_SIZE];
    int32_t status;

    /* Initialize a to sample */
    strcpy(a, SAMPLE_STRING);
    strcpy(b, "");

    status = IecStringCopy(a, sizeof(a), b);

    TEST_ASSERT_EQUAL_STRING("", a);
    TEST_ASSERT_EQUAL_INT(LIBRARY_ERROR_NONE, status);

    TEST_DONE;
}

_TEST test_copy_size_1(void) {
    char a[SAMPLE_SIZE], b[SAMPLE_SIZE];
    int32_t status;

    /* Initialize a to sample */
    strcpy(a, SAMPLE_STRING);
    strcpy(b, SAMPLE_STRING);

    status = IecStringCopy(a, 1, b);

    TEST_ASSERT_EQUAL_STRING("", a);
    TEST_ASSERT_EQUAL_INT(IECSTRING_WARNING_TRUNCATE, status);

    TEST_DONE;
}

_TEST test_copy_size_large(void) {
    char a[LARGE_SIZE], b[LARGE_SIZE];
    int32_t status;

    /* Initialize b */
    memset(b, 'z', LARGE_SIZE - 1);
    b[LARGE_SIZE - 1] = '\0';

    status = IecStringCopy(a, sizeof(a), b);

    TEST_ASSERT_EQUAL_STRING(b, a);
    TEST_ASSERT_EQUAL_INT(LIBRARY_ERROR_NONE, status);

    TEST_DONE;
}

_TEST test_copy_null_source(void) {
    char a[SAMPLE_SIZE];
    int32_t status;

    strcpy(a, SAMPLE_STRING);

    status = IecStringCopy(a, sizeof(a), NULL);

    TEST_ASSERT_EQUAL_STRING(SAMPLE_STRING, a);
    TEST_ASSERT_EQUAL_INT(IECSTRING_ERROR_NULL, status);

    TEST_DONE;
}

_TEST test_copy_null_destination(void) {
    char b[SAMPLE_SIZE];
    int32_t status;

    strcpy(b, SAMPLE_STRING);

    status = IecStringCopy(NULL, SAMPLE_SIZE, b);

    TEST_ASSERT_EQUAL_INT(IECSTRING_ERROR_NULL, status);

    TEST_DONE;
}

_TEST test_copy_size_zero(void) {
    char a[SAMPLE_SIZE], b[SAMPLE_SIZE];
    int32_t status;

    /* Initialize a to sample */
    strcpy(a, SAMPLE_STRING);

    status = IecStringCopy(a, 0, b);

    TEST_ASSERT_EQUAL_STRING(SAMPLE_STRING, a);
    TEST_ASSERT_EQUAL_INT(IECSTRING_ERROR_SIZE, status);

    TEST_DONE;
}

_TEST test_copy_overlap_destination(void) {
    char a[SAMPLE_SIZE];
    char* b;
    int32_t status;

    /* Initialize a to sample */
    strcpy(a, SAMPLE_STRING);
    /* Assign source to overlap destination */
    b = a + sizeof(SAMPLE_STRING) / 2;

    status = IecStringCopy(a, sizeof(a), b);

    TEST_ASSERT_EQUAL_STRING(SAMPLE_STRING, a);
    TEST_ASSERT_EQUAL_INT(IECSTRING_ERROR_OVERLAP, status);

    TEST_DONE;
}

_TEST test_copy_overlap_source(void) {
    char* a;
    char b[SAMPLE_SIZE];
    char c[SAMPLE_SIZE];
    int32_t status;

    strcpy(b, SAMPLE_STRING);
    /* Assign destination to overlap source */
    a = b + sizeof(SAMPLE_STRING) / 2;
    strcpy(c, a);

    status = IecStringCopy(a, SAMPLE_SIZE / 2, b);

    TEST_ASSERT_EQUAL_STRING(c, a);
    TEST_ASSERT_EQUAL_INT(IECSTRING_ERROR_OVERLAP, status);

    TEST_DONE;
}

_TEST test_copy_truncate(void) {
    char a[11], b[SAMPLE_SIZE];
    int32_t status;

    strcpy(b, "0123456789abc");

    status = IecStringCopy(a, sizeof(a), b);

    TEST_ASSERT_EQUAL_STRING("0123456789", a);
    TEST_ASSERT_EQUAL_INT(IECSTRING_WARNING_TRUNCATE, status);

    TEST_DONE;
}

UNITTEST_FIXTURES(fixtures) {
    new_TestFixture("IecStringCopy from variable", test_copy_variable),
    new_TestFixture("IecStringCopy from literal", test_copy_literal),
    new_TestFixture("IecStringCopy empty source", test_copy_empty_source),
    new_TestFixture("IecStringCopy destination size 1", test_copy_size_1),
    new_TestFixture("IecStringCopy large size", test_copy_size_large),
    new_TestFixture("IecStringCopy null source", test_copy_null_source),
    new_TestFixture("IecStringCopy null destination",
                    test_copy_null_destination),
    new_TestFixture("IecStringCopy zero size", test_copy_size_zero),
    new_TestFixture("IecStringCopy overlap destination",
                    test_copy_overlap_destination),
    new_TestFixture("IecStringCopy overlap source", test_copy_overlap_source),
    new_TestFixture("IecStringCopy truncate", test_copy_truncate)
};

UNITTEST_CALLER_TEST (copy_set, "IecStringCopy test set", fixtures);
```

#### test_concat.c - Test IecStringConcat
```c
#include <UnitTest.h>
#include <IecString.h>
#include <stdint.h>
#include <string.h>

#define SAMPLE_STRING_START "Hello"
#define SAMPLE_STRING_END " World!"
#define SAMPLE_SIZE 81
#define LIBRARY_ERROR_NONE 0
#define LARGE_SIZE 1001

_TEST test_concat_variable(void) {
    char a[SAMPLE_SIZE], b[SAMPLE_SIZE];
    int32_t status;

    strcpy(a, SAMPLE_STRING_START);
    strcpy(b, SAMPLE_STRING_END);

    status = IecStringConcat(a, sizeof(a), b);

    TEST_ASSERT_EQUAL_STRING(SAMPLE_STRING_START SAMPLE_STRING_END, a);
    TEST_ASSERT_EQUAL_INT(LIBRARY_ERROR_NONE, status);

    TEST_DONE;
}

_TEST test_concat_literal(void) {
    char a[SAMPLE_SIZE];
    int32_t status;

    strcpy(a, SAMPLE_STRING_START);

    status = IecStringConcat(a, sizeof(a), SAMPLE_STRING_END);

    TEST_ASSERT_EQUAL_STRING(SAMPLE_STRING_START SAMPLE_STRING_END, a);
    TEST_ASSERT_EQUAL_INT(LIBRARY_ERROR_NONE, status);

    TEST_DONE;
}

_TEST test_concat_size_1(void) {
    char a[SAMPLE_SIZE], b[SAMPLE_SIZE];
    int32_t status;

    strcpy(a, "");
    strcpy(b, SAMPLE_STRING_END);

    status = IecStringConcat(a, 1, b);

    TEST_ASSERT_EQUAL_STRING("", a);
    TEST_ASSERT_EQUAL_INT(IECSTRING_WARNING_TRUNCATE, status);

    TEST_DONE;
}

_TEST test_concat_size_large(void) {
    char a[SAMPLE_SIZE + LARGE_SIZE], b[LARGE_SIZE];
    int32_t status;

    strcpy(a, SAMPLE_STRING_START);

    /* Initialize b */
    memset(b, 'z', LARGE_SIZE - 1);
    b[LARGE_SIZE - 1] = '\0';

    status = IecStringConcat(a, sizeof(a), b);

    /* I don't have a good way to assert this
    if the test runs without crashing, that's good */

    TEST_ASSERT_EQUAL_INT(LIBRARY_ERROR_NONE, status);

    TEST_DONE;
}

_TEST test_concat_size_exact(void) {
    char a[sizeof(SAMPLE_STRING_START) + 10];
    int32_t status;

    strcpy(a, SAMPLE_STRING_START);

    status = IecStringConcat(a, sizeof(a), "0123456789");

    TEST_ASSERT_EQUAL_STRING(SAMPLE_STRING_START "0123456789", a);
    TEST_ASSERT_EQUAL_INT(LIBRARY_ERROR_NONE, status);

    TEST_DONE;
}

_TEST test_concat_size_invalid(void) {
    char a[SAMPLE_SIZE], b[SAMPLE_SIZE];
    int32_t status;

    strcpy(a, SAMPLE_STRING_START);
    strcpy(b, SAMPLE_STRING_END);

    status = IecStringConcat(a, sizeof(SAMPLE_STRING_START) - 1, b);

    TEST_ASSERT_EQUAL_STRING(SAMPLE_STRING_START, a);
    TEST_ASSERT_EQUAL_INT(IECSTRING_ERROR_SIZE, status);

    TEST_DONE;
}

_TEST test_concat_null_source(void) {
    char a[SAMPLE_SIZE];
    int32_t status;

    strcpy(a, SAMPLE_STRING_START);

    status = IecStringConcat(a, sizeof(a), NULL);

    TEST_ASSERT_EQUAL_STRING(SAMPLE_STRING_START, a);
    TEST_ASSERT_EQUAL_INT(IECSTRING_ERROR_NULL, status);

    TEST_DONE;
}

_TEST test_concat_null_destination(void) {
    char b[SAMPLE_SIZE];
    int32_t status;

    strcpy(b, SAMPLE_STRING_END);

    status = IecStringConcat(NULL, SAMPLE_SIZE, b);

    TEST_ASSERT_EQUAL_INT(IECSTRING_ERROR_NULL, status);

    TEST_DONE;
}

_TEST test_concat_size_zero(void) {
    char a[SAMPLE_SIZE], b[SAMPLE_SIZE];
    int32_t status;

    strcpy(a, SAMPLE_STRING_START);
    strcpy(b, SAMPLE_STRING_END);

    status = IecStringConcat(a, 0, b);

    TEST_ASSERT_EQUAL_STRING(SAMPLE_STRING_START, a);
    TEST_ASSERT_EQUAL_INT(IECSTRING_ERROR_SIZE, status);

    TEST_DONE;
}

_TEST test_concat_overlap_destination(void) {
    char a[SAMPLE_SIZE];
    char* b;
    int32_t status;

    strcpy(a, SAMPLE_STRING_START);
    /* Assign source to overlap destination */
    b = a + sizeof(SAMPLE_STRING_START) / 2;

    status = IecStringConcat(a, sizeof(a), b);

    TEST_ASSERT_EQUAL_STRING(SAMPLE_STRING_START, a);
    TEST_ASSERT_EQUAL_INT(IECSTRING_ERROR_OVERLAP, status);

    TEST_DONE;
}

_TEST test_concat_overlap_source(void) {
    char* a;
    char b[SAMPLE_SIZE];
    char c[SAMPLE_SIZE];
    int32_t status;

    strcpy(b, SAMPLE_STRING_END);
    /* Assign destination to overlap source */
    a = b + sizeof(SAMPLE_STRING_END) / 2;
    strcpy(c, a);

    status = IecStringConcat(a, sizeof(a), b);

    TEST_ASSERT_EQUAL_STRING(c, a);
    TEST_ASSERT_EQUAL_INT(IECSTRING_ERROR_OVERLAP, status);

    TEST_DONE;
}

_TEST test_concat_truncate(void) {
    char a[11], b[SAMPLE_SIZE];
    int32_t status;

    strcpy(a, "0123456");
    strcpy(b, "789abc");

    status = IecStringConcat(a, sizeof(a), b);

    TEST_ASSERT_EQUAL_STRING("0123456789", a);
    TEST_ASSERT_EQUAL_INT(IECSTRING_WARNING_TRUNCATE, status);

    TEST_DONE;
}

UNITTEST_FIXTURES(fixtures) {
    new_TestFixture("IecStringConcat from variable", test_concat_variable),
    new_TestFixture("IecStringConcat from literal", test_concat_literal),
    new_TestFixture("IecStringConcat destination size 1", test_concat_size_1),
    new_TestFixture("IecStringConcat large size", test_concat_size_large),
    new_TestFixture("IecStringConcat exact size", test_concat_size_exact),
    new_TestFixture("IecStringConcat invalid size", test_concat_size_invalid),
    new_TestFixture("IecStringConcat null source", test_concat_null_source),
    new_TestFixture("IecStringConcat null destination",
                    test_concat_null_destination),
    new_TestFixture("IecStringConcat size zero", test_concat_size_zero),
    new_TestFixture("IecStringConcat overlap destination",
                    test_concat_overlap_destination),
    new_TestFixture("IecStringConcat overlap source",
                    test_concat_overlap_source),
    new_TestFixture("IecStringConcat truncate", test_concat_truncate)
};

UNITTEST_CALLER_TEST (concat_set, "IecStringConcat test set", fixtures);
```

#### test_compare.c - Test IecStringCompare
```c
#include <UnitTest.h>
#include <IecString.h>
#include <stdint.h>
#include <stdbool.h>
#include <string.h>

#define SIZE_STRING 11
#define STRING_SAMPLE "ABC123"
#define STRING_MATCH "ABC"
#define STRING_NO_MATCH "DEF"

_TEST test_compare_variable(void)
{
    char a[SIZE_STRING], b[SIZE_STRING];
    strcpy(a, STRING_SAMPLE);
    strcpy(b, STRING_MATCH);

    int16_t result = IecStringCompare(a, b, 3);

    /* No modifications to strings */
    TEST_ASSERT_EQUAL_STRING(STRING_SAMPLE, a);
    TEST_ASSERT_EQUAL_STRING(STRING_MATCH, b);
    /* Equal */
    TEST_ASSERT_EQUAL_INT(true, result == 0);

    TEST_DONE;
}

_TEST test_compare_literal(void)
{
    int16_t result = IecStringCompare(STRING_SAMPLE, STRING_MATCH, 4);

    /* Greater than */
    TEST_ASSERT_EQUAL_INT(true, result > 0);

    TEST_DONE;
}

_TEST test_compare_greater(void)
{
    int16_t result = IecStringCompare(STRING_SAMPLE, STRING_MATCH, sizeof(STRING_SAMPLE));

    /* Greater than */
    TEST_ASSERT_EQUAL_INT(true, result > 0);

    TEST_DONE;
}

_TEST test_compare_lesser(void)
{
    int16_t result = IecStringCompare(STRING_SAMPLE, STRING_NO_MATCH, sizeof(STRING_SAMPLE));

    /* Less than */
    TEST_ASSERT_EQUAL_INT(true, result < 0);

    TEST_DONE;
}

_TEST test_compare_equal(void)
{
    int16_t result = IecStringCompare(STRING_MATCH, STRING_MATCH, 3);

    /* Equal */
    TEST_ASSERT_EQUAL_INT(true, result == 0);

    TEST_DONE;
}

_TEST test_compare_extra(void)
{
    int16_t result = IecStringCompare(STRING_MATCH, STRING_MATCH, 4);

    /* Equal */
    TEST_ASSERT_EQUAL_INT(true, result == 0);

    TEST_DONE;
}

_TEST test_compare_zero(void)
{
    int16_t result = IecStringCompare(STRING_SAMPLE, STRING_NO_MATCH, 0);

    /* Equal */
    TEST_ASSERT_EQUAL_INT(true, result == 0);

    TEST_DONE;
}

_TEST test_compare_null_1(void)
{
    int16_t result = IecStringCompare(NULL, STRING_MATCH, 3);

    /* Greater than */
    TEST_ASSERT_EQUAL_INT(true, result < 0);

    TEST_DONE;
}

_TEST test_compare_null_2(void)
{
    int16_t result = IecStringCompare(STRING_SAMPLE, NULL, 3);

    /* Greater than */
    TEST_ASSERT_EQUAL_INT(true, result > 0);

    TEST_DONE;
}

UNITTEST_FIXTURES(fixtures)
{
    new_TestFixture("IecStringCompare from variables", test_compare_variable),
    new_TestFixture("IecStringCompare from literals", test_compare_literal),
    new_TestFixture("IecStringCompare greater than", test_compare_greater),
    new_TestFixture("IecStringCompare less than", test_compare_lesser),
    new_TestFixture("IecStringCompare equal", test_compare_equal),
    new_TestFixture("IecStringCompare extra characters", test_compare_extra),
    new_TestFixture("IecStringCompare zero characters", test_compare_zero),
    new_TestFixture("IecStringCompare null string 1", test_compare_null_1),
    new_TestFixture("IecStringCompare null string 2", test_compare_null_2)
};

UNITTEST_CALLER_TEST (compare_set, "IecStringCompare test set", fixtures);
```

#### test_length.c - Test IecStringLength
```c
#include <UnitTest.h>
#include <IecString.h>
#include <stdint.h>
#include <stdbool.h>
#include <string.h>

#define STRING_SAMPLE "The quick brown fox jumps over the lazy dog"

_TEST test_length_variable(void)
{
    char a[81];
    strcpy(a, STRING_SAMPLE);

    uint32_t length = IecStringLength(a);

    /* No modifications to strings */
    TEST_ASSERT_EQUAL_STRING(STRING_SAMPLE, a);

    TEST_ASSERT_EQUAL_INT(43, length);

    TEST_DONE;
}

_TEST test_length_literal(void)
{
    uint32_t length = IecStringLength(STRING_SAMPLE);

    TEST_ASSERT_EQUAL_INT(43, length);

    TEST_DONE;
}

_TEST test_length_large(void)
{
    char a[10000] = {0};
    memset(a, 'a', 7500);

    uint32_t length = IecStringLength(a);

    TEST_ASSERT_EQUAL_INT(7500, length);

    TEST_DONE;
}

_TEST test_length_null(void)
{
    uint32_t length = IecStringLength(NULL);

    TEST_ASSERT_EQUAL_INT(0, length);

    TEST_DONE;
}

UNITTEST_FIXTURES(fixtures)
{
    new_TestFixture("IecStringLength from variables", test_length_variable),
    new_TestFixture("IecStringLength from literals", test_length_literal),
    new_TestFixture("IecStringLength large legth", test_length_large),
    new_TestFixture("IecStringLength null", test_length_null)
};

UNITTEST_CALLER_TEST (length_set, "IecStringLength test set", fixtures);
```

#### test_first.c - Test IecStringFirst
```c
#include <UnitTest.h>
#include <IecString.h>
#include <stdint.h>
#include <string.h>

#define SIZE_STRING 81
#define SAMPLE_STRING "abcde12345"
#define SAMPLE_MULTIPLE "abc123abc123"

_TEST test_first_variable(void)
{
    char find = '3';
    char a[SIZE_STRING] = SAMPLE_STRING;

    /* Call the function with variable arguments */
    uint32_t address = IecStringFirst(a, (uint8_t)find);

    /* Test the input string has not be modified */
    TEST_ASSERT_EQUAL_STRING(a, SAMPLE_STRING);
    /* Test the result */
    TEST_ASSERT_EQUAL_INT(&a + 8, address);

    TEST_DONE;
}

_TEST test_first_literal(void)
{
    /* Call the function with literal arguments */
    uint32_t address = IecStringFirst(SAMPLE_STRING, (uint8_t)'3');

    /* Test the result */
    TEST_ASSERT_EQUAL_INT(&SAMPLE_STRING + 8, address);

    TEST_DONE;
}

_TEST test_first_first(void)
{
    uint32_t address = IecStringFirst(SAMPLE_STRING, (uint8_t)'a');

    TEST_ASSERT_EQUAL_INT(&SAMPLE_STRING, address);

    TEST_DONE;
}

_TEST test_first_last(void)
{
    uint32_t address = IecStringFirst(SAMPLE_STRING, (uint8_t)'5');

    TEST_ASSERT_EQUAL_INT(&SAMPLE_STRING + strlen(SAMPLE_STRING), address);

    TEST_DONE;
}

_TEST test_first_multiple(void)
{
    uint32_t address = IecStringFirst(SAMPLE_MULTIPLE, (uint8_t)'b');

    TEST_ASSERT_EQUAL_INT(&SAMPLE_MULTIPLE + 1, address);

    TEST_DONE;
}

_TEST test_first_none(void)
{
    uint32_t address = IecStringFirst(SAMPLE_MULTIPLE, (uint8_t)'g');

    TEST_ASSERT_EQUAL_INT(0, address);

    TEST_DONE;
}

/* Test special character */
/* Test non-ascii character */
/* Test null string */

UNITTEST_FIXTURES(fixtures) {
    new_TestFixture("IecStringFirst from variable", test_first_variable),
    new_TestFixture("IecStringFirst from literal", test_first_literal),
    new_TestFixture("IecStringFirst first character", test_first_first),
    new_TestFixture("IecStringFirst last character", test_first_last),
    new_TestFixture("IecStringFirst multiple characters", test_first_multiple),
    new_TestFixture("IecStringFirst zero characters", test_first_none)
};

UNITTEST_CALLER_TEST(first_set, "IecStringFirst test set", fixtures);
```

#### test_last.c - Test IecStringLast
```c
#include <UnitTest.h>
#include <IecString.h>
#include <stdint.h>
#include <string.h>

_TEST test_last_variable(void)
{
    char find = '3';
    char a[] = "abcde12345";

    /* Call the function with variable arguments */
    uint32_t address = IecStringLast(a, find);

    /* Test the input string has not be modified */
    TEST_ASSERT_EQUAL_STRING("abcde12345", a);
    /* Test the result */
    TEST_ASSERT_EQUAL_INT((unsigned)a + 7, address);

    TEST_DONE;
}

_TEST test_last_literal(void)
{
    char a[] = "abcde12345";

    /* Call the function with literal character */
    uint32_t address = IecStringLast(a, '3');

    /* Test the input string has not be modified */
    TEST_ASSERT_EQUAL_STRING("abcde12345", a);
    /* Test the result */
    TEST_ASSERT_EQUAL_INT((unsigned)a + 7, address);

    TEST_DONE;
}

_TEST test_last_first(void)
{
    char a[] = "abcde12345";

    uint32_t address = IecStringLast(a, 'a');

    /* Test the input string has not be modified */
    TEST_ASSERT_EQUAL_STRING("abcde12345", a);
    /* Test the result */
    TEST_ASSERT_EQUAL_INT((unsigned)a , address);

    TEST_DONE;
}

_TEST test_last_last(void)
{
    char a[] = "abcde12345";

    uint32_t address = IecStringLast(a, '5');

    /* Test the input string has not be modified */
    TEST_ASSERT_EQUAL_STRING("abcde12345", a);
    /* Test the result */
    TEST_ASSERT_EQUAL_INT((unsigned)a + 9, address);

    TEST_DONE;
}

_TEST test_last_multiple(void)
{
    char b[] = "abc123abc123";

    uint32_t address = IecStringLast(b, 'b');

    /* Test the input string has not be modified */
    TEST_ASSERT_EQUAL_STRING("abc123abc123", b);
    /* Test the result */
    TEST_ASSERT_EQUAL_INT((unsigned)b + 7, address);

    TEST_DONE;
}

_TEST test_last_many(void)
{
    char c[] = "aaaaa aaaaa";

    uint32_t address = IecStringLast(c, 'a');

    /* Test the input string has not be modified */
    TEST_ASSERT_EQUAL_STRING("aaaaa aaaaa", c);
    /* Test the result */
    TEST_ASSERT_EQUAL_INT((unsigned)c + 10, address);

    TEST_DONE;
}

_TEST test_last_none(void)
{
    char b[] = "abc123abc123";

    uint32_t address = IecStringLast(b, 'g');

    /* Test the input string has not be modified */
    TEST_ASSERT_EQUAL_STRING("abc123abc123", b);
    /* Test the result */
    TEST_ASSERT_EQUAL_INT(0, address);

    TEST_DONE;
}

_TEST test_last_special(void)
{
    char find = 6;
    char a[] = "abcde12345";
    memset(a + 3, find, 1);

    /* Call with special character */
    uint32_t address = IecStringLast(a, find);

    /* Test the result */
    TEST_ASSERT_EQUAL_INT((unsigned)a + 3, address);

    TEST_DONE;
}

_TEST test_last_nonascii(void)
{
    char find = 140;
    char a[] = "abcde12345";
    memset(a + 3, find, 1);

    /* Call with non-ascii character */
    uint32_t address = IecStringLast(a, find);

    /* Test the result */
    TEST_ASSERT_EQUAL_INT((unsigned)a + 3, address);

    TEST_DONE;
}

_TEST test_last_empty(void)
{
    char a[] = "";

    /* Call with empty string */
    uint32_t address = IecStringLast(a, '3');

    /* Test the result */
    TEST_ASSERT_EQUAL_INT(0, address);

    TEST_DONE;
}

_TEST test_last_null(void)
{
    /* Call with null string */
    uint32_t address = IecStringLast(NULL, '3');

    /* Test the result */
    TEST_ASSERT_EQUAL_INT(0, address);

    TEST_DONE;
}

UNITTEST_FIXTURES(fixtures) {
    new_TestFixture("IecStringLast from variable", test_last_variable),
    new_TestFixture("IecStringLast from literal", test_last_literal),
    new_TestFixture("IecStringLast first character", test_last_first),
    new_TestFixture("IecStringLast last character", test_last_last),
    new_TestFixture("IecStringLast multiple characters", test_last_multiple),
    new_TestFixture("IecStringLast many characters", test_last_many),
    new_TestFixture("IecStringLast zero characters", test_last_none),
    new_TestFixture("IecStringLast special character", test_last_special),
    new_TestFixture("IecStringLast non-ascii character", test_last_nonascii),
    new_TestFixture("IecStringLast empty string", test_last_empty),
    new_TestFixture("IecStringLast null string", test_last_null)
};

UNITTEST_CALLER_TEST(last_set, "IecStringLast test set", fixtures);
```

#### test_find.c - Test IecStringFind
```c
#include <UnitTest.h>
#include <IecString.h>
#include <stdint.h>
#include <string.h>

#define STRING_SAMPLE "The quick brown fox jumps over the lazy dog"

_TEST test_find_variable(void)
{
    char a[] = STRING_SAMPLE;
    char find[] = "fox";

    /* Call the function with variable arguments */
    uint32_t address = IecStringFind(a, find);

    /* Test the input string has not be modified */
    TEST_ASSERT_EQUAL_STRING(STRING_SAMPLE, a);
    /* Test the result */
    TEST_ASSERT_EQUAL_INT((unsigned)a + 16, address);

    TEST_DONE;
}

_TEST test_find_literal(void)
{
    char a[] = STRING_SAMPLE;

    /* Call the function with variable arguments */
    uint32_t address = IecStringFind(a, "fox");

    /* Test the input string has not be modified */
    TEST_ASSERT_EQUAL_STRING(STRING_SAMPLE, a);
    /* Test the result */
    TEST_ASSERT_EQUAL_INT((unsigned)a + 16, address);

    TEST_DONE;
}

_TEST test_find_single(void)
{
    char a[] = STRING_SAMPLE;

    /* Call the function with variable arguments */
    uint32_t address = IecStringFind(a, "k");

    /* Test the input string has not be modified */
    TEST_ASSERT_EQUAL_STRING(STRING_SAMPLE, a);
    /* Test the result */
    TEST_ASSERT_EQUAL_INT((unsigned)a + 8, address);

    TEST_DONE;
}

UNITTEST_FIXTURES(fixtures) {
    new_TestFixture("IecStringFind from variable", test_find_variable),
    new_TestFixture("IecStringFind from literal", test_find_literal),
    new_TestFixture("IecStringFind single character", test_find_single)
};

UNITTEST_CALLER_TEST(find_set, "IecStringFind test set", fixtures);
```

#### test_first_in.c - Test IecStringFirstIn
```c
#include <UnitTest.h>
#include <IecString.h>
#include <stdint.h>
#include <string.h>

_TEST test_first_in_literal(void)
{
    char a[] = "abcd4321";

    /* Call function */
    uint32_t address = IecStringFirstIn(a, "0123456789");

    /* Test immutability */
    TEST_ASSERT_EQUAL_STRING("abcd4321", a);
    /* Test result */
    TEST_ASSERT_EQUAL_INT((unsigned)a + 4, address);

    TEST_DONE;
}

UNITTEST_FIXTURES(fixtures) {
    new_TestFixture("IecStringFirstIn from literal", test_first_in_literal)
};

UNITTEST_CALLER_TEST(first_in_set, "IecStringFirstIn test set", fixtures);
```

#### test_length_in.c - Test IecStringLengthIn
```c
#include <UnitTest.h>
#include <IecString.h>
#include <stdint.h>
#include <string.h>

_TEST test_length_in_literal(void)
{
    char a[] = "4321abcd";

    /* Call function */
    uint32_t length = IecStringLengthIn(a, "0123456789");

    /* Test immutability */
    TEST_ASSERT_EQUAL_STRING("4321abcd", a);
    /* Test result */
    TEST_ASSERT_EQUAL_INT(4, length);

    TEST_DONE;
}

UNITTEST_FIXTURES(fixtures) {
    new_TestFixture("IecStringLengthIn from literal", test_length_in_literal)
};

UNITTEST_CALLER_TEST(length_in_set, "IecStringLengthIn test set", fixtures);
```

#### test_start.c - Test IecStringStartsWith
```c
#include <UnitTest.h>
#include <IecString.h>
#include <stdint.h>
#include <stdbool.h>
#include <string.h>

#define SIZE_STRING 11
#define STRING_SAMPLE_GREATER "ABC123"
#define STRING_SAMPLE_EQUAL "ABC"
#define STRING_SAMPLE_LESSER "AB"
#define STRING_MATCH "ABC"
#define STRING_NO_MATCH "DEF"

_TEST test_start_variable(void)
{
    char a[SIZE_STRING], b[SIZE_STRING];
    strcpy(a, STRING_SAMPLE_GREATER);
    strcpy(b, STRING_MATCH);

    uint8_t result = IecStringStartsWith(a, b);

    /* No modifications to strings */
    TEST_ASSERT_EQUAL_STRING(STRING_SAMPLE_GREATER, a);
    TEST_ASSERT_EQUAL_STRING(STRING_MATCH, b);
    /* Match */
    TEST_ASSERT_EQUAL_INT(true, result);

    TEST_DONE;
}

_TEST test_start_literal(void)
{
    uint8_t result = IecStringStartsWith(STRING_SAMPLE_GREATER, STRING_MATCH);

    TEST_ASSERT_EQUAL_INT(true, result);

    TEST_DONE;
}

_TEST test_start_equal_match(void)
{
    uint8_t result = IecStringStartsWith(STRING_SAMPLE_EQUAL, STRING_MATCH);

    TEST_ASSERT_EQUAL_INT(true, result);

    TEST_DONE;
}

_TEST test_start_greater_no_match(void)
{
    uint8_t result = IecStringStartsWith(STRING_SAMPLE_GREATER, STRING_NO_MATCH);

    TEST_ASSERT_EQUAL_INT(false, result);

    TEST_DONE;
}

_TEST test_start_equal_no_match(void)
{
    uint8_t result = IecStringStartsWith(STRING_SAMPLE_EQUAL, STRING_NO_MATCH);

    TEST_ASSERT_EQUAL_INT(false, result);

    TEST_DONE;
}

_TEST test_start_lesser(void)
{
    uint8_t result = IecStringStartsWith(STRING_SAMPLE_LESSER, STRING_MATCH);

    TEST_ASSERT_EQUAL_INT(false, result);

    TEST_DONE;
}

_TEST test_start_null_1(void)
{
    uint8_t result = IecStringStartsWith(NULL, STRING_MATCH);

    TEST_ASSERT_EQUAL_INT(false, result);

    TEST_DONE;
}

_TEST test_start_null_2(void)
{
    uint8_t result = IecStringStartsWith(STRING_SAMPLE_GREATER, NULL);

    TEST_ASSERT_EQUAL_INT(false, result);

    TEST_DONE;
}

UNITTEST_FIXTURES(fixtures)
{
    new_TestFixture("IecStringStartsWith from variables", test_start_variable),
    new_TestFixture("IecStringStartsWith from literals", test_start_literal),
    new_TestFixture("IecStringStartsWith equal size match", test_start_equal_match),
    new_TestFixture("IecStringStartsWith greater size no match", test_start_greater_no_match),
    new_TestFixture("IecStringStartsWith equal size no match", test_start_equal_no_match),
    new_TestFixture("IecStringStartsWith lesser size", test_start_lesser),
    new_TestFixture("IecStringStartsWith null string 1", test_start_null_1),
    new_TestFixture("IecStringStartsWith null string 2", test_start_null_2)
};

UNITTEST_CALLER_TEST (start_set, "IecStringStartsWith test set", fixtures);
```

#### test_end.c - Test IecStringEndsWith
```c
#include <UnitTest.h>
#include <IecString.h>
#include <stdint.h>
#include <stdbool.h>
#include <string.h>

#define SIZE_STRING 11
#define STRING_SAMPLE_GREATER "ABC123"
#define STRING_SAMPLE_EQUAL "123"
#define STRING_SAMPLE_LESSER "23"
#define STRING_MATCH "123"
#define STRING_NO_MATCH "456"

_TEST test_end_variable(void)
{
    char a[SIZE_STRING], b[SIZE_STRING];
    strcpy(a, STRING_SAMPLE_GREATER);
    strcpy(b, STRING_MATCH);

    uint8_t result = IecStringEndsWith(a, b);

    /* No modifications to strings */
    TEST_ASSERT_EQUAL_STRING(STRING_SAMPLE_GREATER, a);
    TEST_ASSERT_EQUAL_STRING(STRING_MATCH, b);
    /* Match */
    TEST_ASSERT_EQUAL_INT(true, result);

    TEST_DONE;
}

UNITTEST_FIXTURES(fixtures)
{
    new_TestFixture("IecStringEndsWith from variables", test_end_variable)
};

UNITTEST_CALLER_TEST (end_set, "IecStringEndsWith test set", fixtures);
```

#### test_replace.c - Test IecStringReplace
```c
#include <UnitTest.h>
#include <IecString.h>
#include <string.h>
#include <stdint.h>

_TEST replace_basic(void) {
    char a[81], b[81], f[81], r[81];
    int32_t status;

    strcpy(b, "The quick brown fox");
    strcpy(f, "quick");
    strcpy(r, "slow");

    status = IecStringReplace(a, sizeof(a), b, f, r);

    TEST_ASSERT_EQUAL_STRING("The slow brown fox", a);
    TEST_ASSERT_EQUAL_INT(0, status);

    TEST_DONE;
}

_TEST replace_multiple(void) {
    char a[81], b[81], f[81], r[81];
    int32_t status;

    strcpy(b, "The quick brown fox");
    strcpy(f, " ");
    strcpy(r, "_");

    status = IecStringReplace(a, sizeof(a), b, f, r);

    TEST_ASSERT_EQUAL_STRING("The_quick_brown_fox", a);
    TEST_ASSERT_EQUAL_INT(0, status);

    TEST_DONE;
}

_TEST replace_null_source(void) {
    char a[81], f[81], r[81];
    int32_t status;

    strcpy(a, "Test");

    status = IecStringReplace(a, sizeof(a), f, r, NULL);

    TEST_ASSERT_EQUAL_STRING("Test", a);
    TEST_ASSERT_EQUAL_INT(IECSTRING_ERROR_NULL, status);

    TEST_DONE;
}

_TEST replace_null_find(void) {
    char a[81], b[81], r[81];
    int32_t status;

    strcpy(a, "Test");

    status = IecStringReplace(a, sizeof(a), NULL, r, b);

    TEST_ASSERT_EQUAL_STRING("Test", a);
    TEST_ASSERT_EQUAL_INT(IECSTRING_ERROR_NULL, status);

    TEST_DONE;
}

_TEST replace_null_replace(void) {
    char a[81], b[81], f[81];
    int32_t status;

    strcpy(a, "Test");

    status = IecStringReplace(a, sizeof(a), f, NULL, b);

    TEST_ASSERT_EQUAL_STRING("Test", a);
    TEST_ASSERT_EQUAL_INT(IECSTRING_ERROR_NULL, status);

    TEST_DONE;
}

_TEST replace_null_destination(void) {
    char b[81], f[81], r[81];
    int32_t status;

    status = IecStringReplace(NULL, 11, b, f, r);

    TEST_ASSERT_EQUAL_INT(IECSTRING_ERROR_NULL, status);

    TEST_DONE;
}

_TEST replace_size(void) {
    char a[81], b[81], f[81], r[81];
    int32_t status;

    strcpy(a, "Test");
    strcpy(b, "The quick brown fox");
    strcpy(f, "quick");
    strcpy(r, "slow");

    status = IecStringReplace(a, 0, b, f, r);

    TEST_ASSERT_EQUAL_STRING("Test", a);
    TEST_ASSERT_EQUAL_INT(IECSTRING_ERROR_SIZE_ZERO, status);

    TEST_DONE;
}

_TEST replace_overlap_source(void) {
    char a[81], f[81], r[81];
    int32_t status;

    strcpy(a, "Test");

    status = IecStringReplace(a, sizeof(a), f, r, a + 1);

    TEST_ASSERT_EQUAL_STRING("Test", a);
    TEST_ASSERT_EQUAL_INT(IECSTRING_ERROR_OVERLAP, status);

    TEST_DONE;
}

_TEST replace_overlap_find(void) {
    char a[81], b[81], r[81];
    int32_t status;

    strcpy(a, "Test");

    status = IecStringReplace(a, sizeof(a), a + 1, r, b);

    TEST_ASSERT_EQUAL_STRING("Test", a);
    TEST_ASSERT_EQUAL_INT(IECSTRING_ERROR_OVERLAP, status);

    TEST_DONE;
}

_TEST replace_overlap_replace(void) {
    char a[81], b[81], f[81];
    int32_t status;

    strcpy(a, "Test");

    status = IecStringReplace(a, sizeof(a), f, a + 1, b);

    TEST_ASSERT_EQUAL_STRING("Test", a);
    TEST_ASSERT_EQUAL_INT(IECSTRING_ERROR_OVERLAP, status);

    TEST_DONE;
}

_TEST replace_truncate(void) {
    char a[11], b[81], f[81], r[81];
    int32_t status;

    strcpy(b, "The quick brown fox");
    strcpy(f, "quick");
    strcpy(r, "slow");

    status = IecStringReplace(a, sizeof(a), b, f, r);

    TEST_ASSERT_EQUAL_STRING("The slow b", a);
    TEST_ASSERT_EQUAL_INT(IECSTRING_WARNING_TRUNCATE, status);

    TEST_DONE;
}

UNITTEST_FIXTURES(fixtures) {
    new_TestFixture("IecStringReplace basic", replace_basic),
    new_TestFixture("IecStringReplace multiple", replace_multiple),
    new_TestFixture("IecStringReplace null source", replace_null_source),
    new_TestFixture("IecStringReplace null find", replace_null_find),
    new_TestFixture("IecStringReplace null replace", replace_null_replace),
    new_TestFixture("IecStringReplace null destination", replace_null_destination),
    new_TestFixture("IecStringReplace size", replace_size),
    new_TestFixture("IecStringReplace overlap source", replace_overlap_source),
    new_TestFixture("IecStringReplace overlap find", replace_overlap_find),
    new_TestFixture("IecStringReplace overlap replace", replace_overlap_replace),
    new_TestFixture("IecStringReplace truncate", replace_truncate)
};

UNITTEST_CALLER_TEST (replace_set, "IecStringReplace test set", fixtures);
```

#### test_split.c - Test IecStringSplit
```c
#include <UnitTest.h>
#include <IecString.h>
#include <stdint.h>
#include <string.h>

_TEST test_split_variable(void)
{
    char a[] = "The quick brown fox jumps over the lazy dog";
    char delimeters[] = " ";
    char b[5][10] = {{0}};
    int32_t result[5] = {0};
    char *address = a, *next_address = 0;
    int i = 0;

    /* Call the function with variable arguments */
    do
    {
        result[i] = IecStringSplit(b[i], sizeof(b[i]), address, delimeters,
                                   (uint32_t*)&next_address);
        address = next_address;
    }
    while (++i < 5 && next_address);

    TEST_ASSERT_EQUAL_STRING("The quick brown fox jumps over the lazy dog", a);

    TEST_ASSERT_EQUAL_STRING("The", b[0]);
    TEST_ASSERT_EQUAL_STRING("quick", b[1]);
    TEST_ASSERT_EQUAL_STRING("brown", b[2]);
    TEST_ASSERT_EQUAL_STRING("fox", b[3]);
    TEST_ASSERT_EQUAL_STRING("jumps", b[4]);

    TEST_ASSERT_EQUAL_INT(IECSTRING_ERROR_NONE, result[0]);
    TEST_ASSERT_EQUAL_INT(IECSTRING_ERROR_NONE, result[1]);
    TEST_ASSERT_EQUAL_INT(IECSTRING_ERROR_NONE, result[2]);
    TEST_ASSERT_EQUAL_INT(IECSTRING_ERROR_NONE, result[3]);
    TEST_ASSERT_EQUAL_INT(IECSTRING_ERROR_NONE, result[4]);

    TEST_DONE;
}

_TEST test_split_multiple(void)
{
    char a[] = "... Apple, Banana, Orange, ...";
    char delimeters[] = " ,.";
    char b[3][10] = {{0}};
    int32_t result[3] = {0};
    char *address = a, *next_address = 0;
    int i = 0;

    /* Call the function with variable arguments */
    do
    {
        result[i] = IecStringSplit(b[i], sizeof(b[i]), address, delimeters,
                                   (uint32_t*)&next_address);
        address = next_address;
    }
    while (++i < 3 && next_address);

    TEST_ASSERT_EQUAL_STRING("... Apple, Banana, Orange, ...", a);

    TEST_ASSERT_EQUAL_STRING("Apple", b[0]);
    TEST_ASSERT_EQUAL_STRING("Banana", b[1]);
    TEST_ASSERT_EQUAL_STRING("Orange", b[2]);

    TEST_ASSERT_EQUAL_INT(IECSTRING_ERROR_NONE, result[0]);
    TEST_ASSERT_EQUAL_INT(IECSTRING_ERROR_NONE, result[1]);
    TEST_ASSERT_EQUAL_INT(IECSTRING_ERROR_NONE, result[2]);

    TEST_DONE;
}

_TEST test_split_truncate(void)
{
    char a[] = "Three, two, one";
    char delimeters[] = " ,";
    char b[4];
    char *next_address;
    int32_t result;

    /* Call the function */
    result = IecStringSplit(b, sizeof(b), a, delimeters, (uint32_t*)&next_address);

    TEST_ASSERT_EQUAL_STRING("Three, two, one", a);

    TEST_ASSERT_EQUAL_STRING("Thr", b);

    TEST_ASSERT_EQUAL_INT(IECSTRING_WARNING_TRUNCATE, result);

    TEST_DONE;
}

UNITTEST_FIXTURES(fixtures) {
    new_TestFixture("IecStringSplit from variable", test_split_variable),
    new_TestFixture("IecStringSplit multiple delimeters", test_split_multiple),
    new_TestFixture("IecStringSplit truncate output", test_split_truncate)
};

UNITTEST_CALLER_TEST(split_set, "IecStringSplit test set", fixtures);
```

#### test_format.c - Test IecStringFormat
```c
#include <UnitTest.h>
#include <IecString.h>
#include <string.h>
#include <stdint.h>
#include <stdbool.h>

#define SAMPLE_SIZE 81
#define SAMPLE_STRING "Hello World!"
#define LIBRARY_ERROR_NONE 0

_TEST format_from_variable(void) {
    char a[SAMPLE_SIZE], b[SAMPLE_SIZE];
    IecStringFormatType args;
    int32_t status;

    strcpy(b, "Error: %b, Temp: %f C, Step: %i, Message: %s");
    args.b[0] = true;
    args.f[0] = 123.456;
    args.i[0] = 15;
    strcpy(args.s[0], "All clear");

    status = IecStringFormat(a, sizeof(a), b, &args);

    TEST_ASSERT_EQUAL_STRING("Error: TRUE, Temp: 123.456000 C, Step: 15, Message: All clear", a);
    TEST_ASSERT_EQUAL_INT(LIBRARY_ERROR_NONE, status);

    TEST_DONE;
}

_TEST format_from_literal(void) {
    char a[SAMPLE_SIZE];
    IecStringFormatType args;
    int32_t status;

    args.b[0] = true;
    args.f[0] = 123.456;
    args.i[0] = 15;
    strcpy(args.s[0], "All clear");

    status = IecStringFormat(a, sizeof(a),
                             "Error: %b, Temp: %f C, Step: %i, Message: %s",
                             &args);

    TEST_ASSERT_EQUAL_STRING("Error: TRUE, Temp: 123.456000 C, Step: 15, Message: All clear", a);
    TEST_ASSERT_EQUAL_INT(LIBRARY_ERROR_NONE, status);

    TEST_DONE;
}

_TEST format_bool(void) {
    char a[SAMPLE_SIZE];
    IecStringFormatType args;
    int32_t status;

    args.b[0] = true;
    args.b[1] = false;
    args.b[2] = 100;
    args.b[3] = false;
    args.b[4] = true;
    args.b[5] = false;

    status = IecStringFormat(a, sizeof(a),
                             "%b, %b, %b, %b, %b, %b, %b", &args);

    TEST_ASSERT_EQUAL_STRING("TRUE, FALSE, TRUE, FALSE, TRUE, FALSE, ", a);
    TEST_ASSERT_EQUAL_INT(LIBRARY_ERROR_NONE, status);

    TEST_DONE;
}

_TEST format_float(void) {
    char a[SAMPLE_SIZE];
    IecStringFormatType args;
    int32_t status;

    args.f[0] = 123456;
    args.f[1] = 2e34;
    args.f[2] = -567890;
    args.f[3] = 1.234567;
    args.f[4] = -1e23;
    args.f[5] = 0;

    status = IecStringFormat(a, sizeof(a),
                             "%f, %f, %f, %f, %f, %f, %f", &args);

    TEST_ASSERT_EQUAL_STRING("123456.000000, 2.000000e+34, -567890.000000, 1.234567, -1.000000e+23, 0, ", a);
    TEST_ASSERT_EQUAL_INT(LIBRARY_ERROR_NONE, status);

    TEST_DONE;
}

_TEST format_int(void) {
    char a[SAMPLE_SIZE];
    IecStringFormatType args;
    int32_t status;

    args.i[0] = -123;
    args.i[1] = INT32_MAX;
    args.i[2] = INT32_MIN;
    args.i[3] = UINT32_MAX;
    args.i[4] = 2147483648U;
    args.i[5] = 0;

    status = IecStringFormat(a, sizeof(a), "%i, %i, %i, %i, %i, %i, %i", &args);

    TEST_ASSERT_EQUAL_STRING("-123, 2147483647, -2147483648, -1, -2147483648, 0, ", a);
    TEST_ASSERT_EQUAL_INT(LIBRARY_ERROR_NONE, status);

    TEST_DONE;
}

_TEST format_string(void) {
    char a[SAMPLE_SIZE];
    IecStringFormatType args;
    int32_t status;

    strcpy(args.s[0], "one");
    strcpy(args.s[1], "two");
    strcpy(args.s[2], "three");
    strcpy(args.s[3], "apple");
    strcpy(args.s[4], "banana");
    strcpy(args.s[5], "carrot");

    status = IecStringFormat(a, sizeof(a), "%s, %s, %s, %s, %s, %s, %s", &args);

    TEST_ASSERT_EQUAL_STRING("one, two, three, apple, banana, carrot, ", a);
    TEST_ASSERT_EQUAL_INT(LIBRARY_ERROR_NONE, status);

    TEST_DONE;
}

_TEST format_null_source(void) {
    char a[SAMPLE_SIZE];
    IecStringFormatType args;
    int32_t status;

    strcpy(a, SAMPLE_STRING);

    status = IecStringFormat(a, sizeof(a), NULL, &args);

    TEST_ASSERT_EQUAL_STRING(SAMPLE_STRING, a);
    TEST_ASSERT_EQUAL_INT(IECSTRING_ERROR_NULL, status);

    TEST_DONE;
}

_TEST format_null_destination(void) {
    char b[SAMPLE_SIZE];
    IecStringFormatType args;
    int32_t status;

    status = IecStringFormat(NULL, SAMPLE_SIZE, b, &args);

    TEST_ASSERT_EQUAL_INT(IECSTRING_ERROR_NULL, status);

    TEST_DONE;
}

_TEST format_null_values(void) {
    char a[SAMPLE_SIZE], b[SAMPLE_SIZE];
    int32_t status;

    strcpy(a, "abc123");
    strcpy(b, SAMPLE_STRING);

    status = IecStringFormat(a, sizeof(a), b, NULL);

    TEST_ASSERT_EQUAL_STRING(SAMPLE_STRING, a);
    TEST_ASSERT_EQUAL_INT(IECSTRING_ERROR_NULL, status);

    TEST_DONE;
}

_TEST format_size_zero(void) {
    char a[SAMPLE_SIZE], b[SAMPLE_SIZE];
    IecStringFormatType args;
    int32_t status;

    strcpy(a, SAMPLE_STRING);

    status = IecStringFormat(a, 0, b, &args);

    TEST_ASSERT_EQUAL_STRING(SAMPLE_STRING, a);
    TEST_ASSERT_EQUAL_INT(IECSTRING_ERROR_SIZE_ZERO, status);

    TEST_DONE;
}

_TEST format_size_1(void) {
    char a[SAMPLE_SIZE], b[SAMPLE_SIZE];
    IecStringFormatType args;
    int32_t status;

    strcpy(b, SAMPLE_STRING);

    status = IecStringFormat(a, 1, b, &args);

    TEST_ASSERT_EQUAL_STRING("", a);
    TEST_ASSERT_EQUAL_INT(IECSTRING_WARNING_TRUNCATE, status);

    TEST_DONE;
}

_TEST format_size_exact_middle(void) {
    char a[20];
    IecStringFormatType args;
    int32_t status;

    strcpy(args.s[0], "quick");

    status = IecStringFormat(a, sizeof(a), "The %s brown fox", &args);

    TEST_ASSERT_EQUAL_STRING("The quick brown fox", a);
    TEST_ASSERT_EQUAL_INT(LIBRARY_ERROR_NONE, status);

    TEST_DONE;
}

_TEST format_size_exact_end(void) {
    char a[20];
    IecStringFormatType args;
    int32_t status;

    strcpy(args.s[0], "fox");

    status = IecStringFormat(a, sizeof(a), "The quick brown %s", &args);

    TEST_ASSERT_EQUAL_STRING("The quick brown fox", a);
    TEST_ASSERT_EQUAL_INT(LIBRARY_ERROR_NONE, status);

    TEST_DONE;
}

_TEST format_overlap_source(void) {
    char *a, b[SAMPLE_SIZE];
    IecStringFormatType args;
    int32_t status;

    strcpy(b, SAMPLE_STRING);
    a = b + 1;

    status = IecStringFormat(a, SAMPLE_SIZE, b, &args);

    TEST_ASSERT_EQUAL_STRING(SAMPLE_STRING, b);
    TEST_ASSERT_EQUAL_INT(IECSTRING_ERROR_OVERLAP, status);

    TEST_DONE;
}

_TEST format_overlap_destination(void) {
    char a[SAMPLE_SIZE], *b;
    IecStringFormatType args;
    int32_t status;

    strcpy(a, SAMPLE_STRING);
    b = a + 1;

    status = IecStringFormat(a, sizeof(a), b, &args);

    TEST_ASSERT_EQUAL_STRING(SAMPLE_STRING, a);
    TEST_ASSERT_EQUAL_INT(IECSTRING_ERROR_OVERLAP, status);

    TEST_DONE;
}

_TEST format_truncate(void) {
    char a[12];
    IecStringFormatType args;
    int32_t status;

    strcpy(args.s[0], "one");
    strcpy(args.s[1], "two");
    strcpy(args.s[2], "three");

    status = IecStringFormat(a, sizeof(a), "%s, %s, %s", &args);

    TEST_ASSERT_EQUAL_STRING("one, two, t", a);
    TEST_ASSERT_EQUAL_INT(IECSTRING_WARNING_TRUNCATE, status);

    TEST_DONE;
}

UNITTEST_FIXTURES(fixtures){
    new_TestFixture("IecStringFormat from variable", format_from_variable),
    new_TestFixture("IecStringFormat from literal", format_from_literal),
    new_TestFixture("IecStringFormat bool", format_bool),
    new_TestFixture("IecStringFormat float", format_float),
    new_TestFixture("IecStringFormat integer", format_int),
    new_TestFixture("IecStringFormat string", format_string),
    new_TestFixture("IecStringFormat null source", format_null_source),
    new_TestFixture("IecStringFormat null destination",
                    format_null_destination),
    new_TestFixture("IecStringFormat null values", format_null_values),
    new_TestFixture("IecStringFormat size zero", format_size_zero),
    new_TestFixture("IecStringFormat size 1", format_size_1),
    new_TestFixture("IecStringFormat size exact format middle",
                    format_size_exact_middle),
    new_TestFixture("IecStringFormat size exact format end",
                    format_size_exact_end),
    new_TestFixture("IecStringFormat overlap source", format_overlap_source),
    new_TestFixture("IecStringFormat overlap destination",
                    format_overlap_destination),
    new_TestFixture("IecStringFormat truncate", format_truncate)
};

UNITTEST_CALLER_TEST (format_set, "IecStringFormat test set", fixtures);
```

#### test_decimal.c - Test IecStringDecimal
```c
#include <UnitTest.h>
#include <IecString.h>
#include <string.h>
#include <stdint.h>

_TEST test_decimal_zeros(void) {
    char a[81];
    int32_t number, status;

    number = 1234;

    status = IecStringDecimal(a, sizeof(a), number, 6, IECSTRING_FLAG_NONE);

    TEST_ASSERT_EQUAL_STRING("001234", a);
    TEST_ASSERT_EQUAL_INT(0, status);

    TEST_DONE;
}

_TEST test_decimal_spaces(void) {
    char a[81];
    int32_t number, status;

    number = -5678;

    status = IecStringDecimal(a, sizeof(a), number, 6, IECSTRING_FLAG_SPACES);

    /* Width includes sign */
    TEST_ASSERT_EQUAL_STRING("- 5678", a);
    TEST_ASSERT_EQUAL_INT(0, status);

    /* Defaults to spaces */
    status = IecStringDecimal(a, sizeof(a), number, 6, IECSTRING_FLAG_SPACES);

    TEST_ASSERT_EQUAL_STRING("- 5678", a);
    TEST_ASSERT_EQUAL_INT(0, status);

    TEST_DONE;
}

_TEST test_decimal_sign_pos(void) {
    char a[81];
    int32_t status;

    status = IecStringDecimal(a, sizeof(a), 123456, 8, IECSTRING_FLAG_SIGN);

    TEST_ASSERT_EQUAL_STRING("+0123456", a);
    TEST_ASSERT_EQUAL_INT(0, status);

    TEST_DONE;
}

_TEST test_decimal_max(void) {
    char a[81];
    int32_t number, status;

    number = INT32_MAX;

    status = IecStringDecimal(a, sizeof(a), number, 0, IECSTRING_FLAG_NONE);

    TEST_ASSERT_EQUAL_STRING("2147483647", a);
    TEST_ASSERT_EQUAL_INT(0, status);

    TEST_DONE;
}

_TEST test_decimal_min(void) {
    char a[81];
    int32_t number, status;

    number = INT32_MIN;

    status = IecStringDecimal(a, sizeof(a), number, 0, IECSTRING_FLAG_NONE);

    TEST_ASSERT_EQUAL_STRING("-2147483648", a);
    TEST_ASSERT_EQUAL_INT(0, status);

    TEST_DONE;
}

_TEST test_decimal_size(void) {
    char a[6];
    int32_t number, status;

    strcpy(a, "abc");
    number = 123456;

    status = IecStringDecimal(a, sizeof(a), number, 0, IECSTRING_FLAG_NONE);

    TEST_ASSERT_EQUAL_STRING("abc", a);
    TEST_ASSERT_EQUAL_INT(IECSTRING_ERROR_SIZE_INVALID, status);

    TEST_DONE;
}

_TEST test_decimal_null(void) {
    int32_t number, status;

    number = 123456;

    status = IecStringDecimal(NULL, 7, number, 0, IECSTRING_FLAG_NONE);

    TEST_ASSERT_EQUAL_INT(IECSTRING_ERROR_NULL, status);

    TEST_DONE;
}

UNITTEST_FIXTURES(fixtures) {
    new_TestFixture("IecStringDecimal zeros", test_decimal_zeros),
    new_TestFixture("IecStringDecimal spaces", test_decimal_spaces),
    new_TestFixture("IecStringDecimal sign positive", test_decimal_sign_pos),
    new_TestFixture("IecStringDecimal max", test_decimal_max),
    new_TestFixture("IecStringDecimal min", test_decimal_min),
    new_TestFixture("IecStringDecimal size error", test_decimal_size),
    new_TestFixture("IecStringDecimal null error", test_decimal_null)
};

UNITTEST_CALLER_TEST (decimal_set, "IecStringDecimal test set", fixtures);
```
